// ---- GlobalTextList.TcGTLO
TEXTLIST GlobalTextList
  90 = '\nTwinSAFE'
  12 = '  %s'
  13 = ' %s'
  153 = ' CH1 Test Pulses Active'
  152 = ' CH1 Test Pulses Not Active'
  154 = ' CH2 Test Pulses Active'
  155 = ' CH2 Test Pulses Not Active'
  157 = ' CH3 Test Pulses Active'
  156 = ' CH3 Test Pulses Not Active'
  221 = ' CH32 Test Pulses Not Active'
  159 = ' CH4 Test Pulses Active'
  158 = ' CH4 Test Pulses Not Active'
  222 = ' CH43 Test Pulses Active'
  223 = ' CH5 Test Pulses Active'
  224 = ' CH5 Test Pulses Not Active'
  225 = ' CH6 Test Pulses Active'
  226 = ' CH6 Test Pulses Not Active'
  227 = ' CH7 Test Pulses Active'
  228 = ' CH7 Test Pulses Not Active'
  229 = ' CH8 Test Pulses Active'
  230 = ' CH8 Test Pulses Not Active'
  283 = ' Connections: %s'
  376 = ' CX HW Date: %s'
  374 = ' CX HW Serial#: %s'
  375 = ' CX HW Sn: %s'
  377 = ' CX HW Vers: %s'
  379 = ' CX Image Level: %s'
  378 = ' CX Image Vers: %s'
  373 = ' CX Serial#: %s'
  372 = ' CX: %s'
  286 = ' Groups: %s'
  150 = ' Logic CH1 and CH2: %s'
  151 = ' Logic CH3 and CH4: %s'
  231 = ' Logic CH5 and CH6: %s'
  232 = ' Logic CH7 and CH8: %s'
  143 = ' Mode: %s'
  380 = ' OS Vers: %s'
  371 = ' OS: %s'
  287 = ' Safety FBs: %s'
  43 = '%0.3f'
  363 = '%0i'
  364 = '%0s'
  486 = '%2.1f'
  487 = '%2.1f Hrs'
  362 = '%n'
  365 = '%N'
  11 = '%s'
  509 = '%s v'
  510 = '%sV'
  539 = '(3.300 v Nominal'
  109 = '(3.300 v Nominal)'
  295 = '(5.000 v Nominal)'
  599 = '(ISO 8601) YYYY-MM-DDThh:mm:ss.sTZD'
  101 = '-- External Supply or cross-circuit --\nTHESE ERRORS ARE ONLY ACTIVE IF\nCurrent Measurement is FALSE'
  102 = '-- External Supply or cross-circuit --\nTHESE ERRORS ARE ONLY VALID IF\nCurrent Measurement ACTIVE is FALSE'
  103 = '-- Open Load, I<20mA, I>500mA --\nTHESE ERRORS ARE ONLY VALID IF\nCurrent Measurement ACTIVE is TRUE'
  503 = '. %s'
  35 = '00%s'
  15 = '1'
  16 = '2'
  190 = '2-CHs Eval Error'
  210 = '2CH\nSync\nVel'
  208 = '2CH\nSync Vel'
  209 = '2CH\nSync Vel &\n2CH Encoder'
  203 = '2CH Eval\nError'
  207 = '2CH Sync Vel'
  49 = '2Channel Eval Error'
  17 = '3'
  18 = '4'
  241 = '5'
  443 = '5s'
  242 = '6'
  243 = '7'
  244 = '8'
  161 = '<17.5v'
  165 = '>30.5v'
  160 = '>30v'
  162 = '>320v'
  163 = '>32v'
  508 = 'Actual'
  496 = 'Actual: %s'
  335 = 'AdditionalLink'
  399 = 'ADS Monitor'
  428 = 'ADS Port: %s'
  28 = 'AND#1'
  26 = 'AND#1 Status'
  30 = 'AND#2'
  406 = 'Applic Name: %s'
  297 = 'AX5000 Drive Safety Option: %s'
  343 = 'AX5206'
  316 = 'AX5206 State: %s'
  296 = 'AX5805'
  269 = 'AX5805 Error'
  270 = 'AX5805 OK'
  294 = 'AX5805 Sn: 00%s'
  317 = 'AX5805 State: %s'
  437 = 'AX5808'
  367 = 'Beckhoff Computer and PLC INFO'
  298 = 'Beckhoff EtherCAT Diagnostics 1'
  319 = 'Beckhoff EtherCAT Diagnostics 2'
  442 = 'Beckhoff EtherCAT Diagostics 1'
  449 = 'Beckhoff EtherCAT Diagostics 2'
  502 = 'BIOS: %s'
  490 = 'Boot Count: %s'
  411 = 'Boot Data Loaded'
  408 = 'Boot Data Loaded: %s'
  326 = 'BootStrap'
  176 = 'C\nH\n \n1'
  180 = 'C\nH\n \n2'
  398 = 'Capturing Data'
  94 = 'CH 1'
  137 = 'Ch 1'
  95 = 'CH 2'
  138 = 'Ch 2'
  96 = 'CH 3'
  139 = 'Ch 3'
  97 = 'CH 4'
  140 = 'Ch 4'
  186 = 'Ch 5'
  187 = 'Ch 6'
  188 = 'Ch 7'
  189 = 'Ch 8'
  47 = 'CH1'
  545 = 'Ch1'
  145 = 'CH1 Test Pulses Active'
  144 = 'CH1 Test Pulses Not Active'
  177 = 'CH2'
  546 = 'Ch2'
  146 = 'CH2 Test Pulses Active'
  147 = 'CH2 Test Pulses Not Active'
  178 = 'CH3'
  547 = 'Ch3'
  549 = 'CH3 Test Pulses Active'
  550 = 'CH3 Test Pulses Not Active'
  179 = 'CH4'
  548 = 'Ch4'
  551 = 'CH4 Test Pulses Active'
  552 = 'CH4 Test Pulses Not Active'
  350 = 'Clear\nCRC Errors'
  368 = 'Clear\nFrames Data'
  351 = 'Clear\nLost Frames'
  352 = 'Clear\nTx/Rx Errors'
  347 = 'Clear CRC Errors'
  348 = 'Clear Lost Frames'
  349 = 'Clear Tx/Rx Errors'
  24 = 'COM'
  5 = 'COM Error'
  463 = 'Computer Hardware Specifics'
  465 = 'Computer Software Specifics'
  387 = "Computer's AMSNetID: %s"
  462 = "Computer's AMSNetIDl: %s"
  386 = "Computer'sAMSNetID: %s"
  369 = 'Computer/Controller Specifics'
  21 = 'Connection 1  (EL1904)'
  435 = 'Connection 1 (EL1904)'
  19 = 'Connection 1 State (EL1904)'
  23 = 'Connection 2  (EL2904)'
  436 = 'Connection 2 (EL2904)'
  292 = 'Connections: %s'
  517 = 'CPU Info'
  122 = 'Current Measurement'
  133 = 'Current Measurement Active'
  134 = 'Current Measurement Not Active'
  126 = 'Current Measurement ON'
  500 = 'Currently: %s'
  482 = 'CX Boot Count: %s'
  459 = 'CX HW Date: %s'
  457 = 'CX HW Sn: %s'
  458 = 'CX HW Vers: %s'
  460 = 'CX Image Level: %s'
  388 = 'CX Image Vers: %s'
  483 = 'CX Oper Time - Days: %s'
  484 = 'CX Oper Time - Hrs: %s'
  485 = 'CX Oper Time: %s Days'
  471 = 'CX Prod Date: %D'
  474 = 'CX Prod Date: %M'
  475 = 'CX Prod Date: %m%d%y'
  473 = 'CX Prod Date: %Mdy'
  476 = 'CX Prod Date: %MM-DD-YYYY'
  470 = 'CX Prod Date: %s'
  472 = 'CX Prod Date: %s Mdy'
  478 = 'CX Prod Date: %t[MM DD YYYY]'
  477 = 'CX Prod Date: %t[MM-DD-YYYY]'
  480 = 'CX Prod Date: %t[MM.dd.YYYY]'
  481 = 'CX Prod Date: %t[MM.dd.yyyy]'
  479 = 'CX Prod Date: %t[MM]-%t[dd]-%t[YYYY]'
  468 = 'CX SN: %s'
  469 = 'CX Type: %s'
  389 = 'CX: %s'
  427 = 'Cycle Count: %s'
  424 = 'Cycle Exceeded'
  426 = 'Cycle Exceeded Flag'
  597 = 'Date/Time Presentation: %s'
  534 = 'Default Gateway: %s'
  181 = 'dfgh'
  529 = 'DHCP Flag'
  22 = 'Diagnostic: %s'
  107 = 'DIP SW: %s'
  106 = 'DIP Switch'
  39 = 'DIP Switch Setting'
  248 = 'E-Stop\nComplete'
  33 = 'EDM'
  441 = 'EDM\nFB Error'
  251 = 'EDM FB\nError'
  342 = 'EK1110'
  315 = 'EK1110 State: %s'
  560 = 'EK1122'
  558 = 'EK1122 State: %s'
  340 = 'EL1004'
  310 = 'EL1004 State: %s'
  451 = 'EL1008'
  445 = 'EL1008 State: %s'
  93 = 'EL1904'
  38 = 'EL1904 DIP Switch Setting'
  264 = 'EL1904 Error'
  8 = 'EL1904 Inputs'
  265 = 'EL1904 OK'
  10 = 'EL1904 puts'
  37 = 'EL1904 Serial Number'
  136 = 'EL1904 Sn: 00%s'
  311 = 'EL1904 State: %s'
  341 = 'EL2004'
  312 = 'EL2004 State: %s'
  444 = 'EL2004 State: 5s'
  452 = 'EL2008'
  446 = 'EL2008 State: %s'
  542 = 'EL2901'
  92 = 'EL2904'
  267 = 'EL2904 Error'
  433 = 'EL2904 Inputs'
  268 = 'EL2904 OK'
  9 = 'EL2904 Outputs'
  70 = 'EL2904 Serial Number'
  108 = 'EL2904 Sn: 00%s'
  313 = 'EL2904 State: %s'
  453 = 'EL3002'
  447 = 'EL3002 State: %s'
  559 = 'EL4032'
  556 = 'EL4032 State: %s'
  454 = 'EL4034'
  448 = 'EL4034 State: %s'
  259 = 'EL6900'
  261 = 'EL6900 Error'
  260 = 'EL6900 OK'
  293 = 'EL6900 Sn: 00%s'
  309 = 'EL6900 State: %s'
  282 = 'EL6930'
  262 = 'EL6930 Error'
  263 = 'EL6930 OK'
  182 = 'EL6930 Sn: 00%s'
  314 = 'EL6930 State: %s'
  455 = 'EL7201 #1'
  456 = 'EL7201 #2'
  557 = 'EL7201 State: %s'
  185 = 'EP1908'
  271 = 'EP1908 Error'
  266 = 'EP1908 OK'
  184 = 'EP1908 Sn: 00%s'
  318 = 'EP1908 State: %s'
  247 = 'Error'
  124 = 'Error Ack Active'
  135 = 'Error Ack Not Active'
  71 = 'Error At The Output'
  72 = 'Error At The Output\nExternal Supply or Cross-Circuit'
  169 = 'Error Clear'
  206 = 'Error In Oper Mode'
  29 = 'EStop'
  430 = 'EStop\nComplete'
  438 = 'EStop\nFB'
  439 = 'EStop\nFB Error'
  250 = 'EStop FB\nError'
  0 = 'EStop Reset'
  344 = 'EtherCAT'
  359 = 'EtherCAT\nDiag1'
  360 = 'EtherCAT\nDiag2'
  345 = 'EtherCAT\nDiagnostic 1'
  346 = 'EtherCAT\nDiagnostic 2'
  299 = 'EtherCAT Master Status and Statistics'
  308 = 'EtherCAT Slaves and Working Counter Status'
  358 = 'EtherCAT Working Counter and Slaves Status'
  100 = 'External Supply or cross-circuit\nTHESE ERRORS ARE ONLY ACTIVE IF\nCurrent Measurement is FALSE'
  99 = 'External Supply or cross-circuit\nTHESE ERRORS ARE ONLY ACTIVE IF '
  415 = 'FALSE'
  25 = 'FB'
  6 = 'FB Error'
  543 = 'Features'
  119 = 'Features:'
  423 = 'First Scan'
  425 = 'First Scan Flag'
  586 = 'For CE Only !'
  585 = 'For CE Only !           !'
  584 = 'For CE Only!'
  355 = 'Frames/Sec: %4.0f'
  304 = 'Frames/Sec: %4.1f'
  353 = 'Frames/Sec: %4f'
  205 = 'Frequency\n> 500Hz'
  518 = 'Frequency: %2.3f'
  523 = 'Frequency: %2.3f GHz'
  291 = 'FW: %s'
  67 = 'Go To'
  69 = 'Go To\nEL1904\nDiagnostics'
  68 = 'Go To\nTwinSAFE\nScreen'
  284 = 'Groups: %s'
  75 = 'HI'
  499 = 'Highest: %s'
  289 = 'HW:'
  290 = 'HW: %s'
  511 = 'In Deg C'
  325 = 'Init'
  331 = 'InitCmdError'
  330 = 'InvVPRS'
  532 = 'IP Address: %s'
  410 = 'Keep Outputs ON BP: %s'
  417 = 'Keep Outputs ON Bypass'
  370 = 'Label'
  422 = 'Last Exec Time (100ns incr): %s'
  516 = 'Last Exec Time (in microsec): %5.1f'
  514 = 'Last Exec Time (in microsec): %5.2f'
  515 = 'Last Exec Time (in microsec): %5.3f'
  513 = 'Last Exec Time (in microsec): %s'
  334 = 'LinkMissing'
  332 = 'LinkNotPresent'
  450 = 'Link_w/o_Com'
  333 = 'Link_w/o_Comm'
  76 = 'LO'
  148 = 'Logic CH1 and CH2: %s'
  149 = 'Logic CH3 and CH4: %s'
  34 = 'Logic Terminal Serial Number'
  305 = 'Lost Frames: %i'
  307 = 'Lost Queued Frames: %i'
  498 = 'Lowest: %s'
  531 = 'MAC Address: %s'
  567 = 'Mainboard'
  571 = 'Mainboard and CPU'
  570 = 'Mainboard Info'
  573 = 'Mainboard, CPU, Memory'
  300 = 'Master: %s'
  277 = 'Max Supply Voltage to MC1 Exceeded'
  278 = 'Max Supply Voltage to MC2 Exceeded'
  541 = 'Maximum Supply Voltage to MC1 Exceeded'
  274 = 'Maximum Temperature Exceeded'
  497 = 'Maximum: %s'
  62 = 'MC Temperatures'
  57 = 'MC Temperatures (in Deg C)'
  112 = 'MC Voltages'
  66 = 'MC Voltages (3.300 v Nominal)'
  54 = 'MC Voltages (3.300v Nominal)'
  540 = 'MC1 Actual Temperature: %0.3f v'
  401 = 'MC1 Actual Temperature: %s C'
  104 = 'MC1 Actual Temperature: %s °C'
  110 = 'MC1 Actual Voltage: %0.3f v'
  84 = 'Mc1 COLD!'
  554 = 'MC1 COLD!'
  77 = 'Mc1 HOT!'
  553 = 'MC1 HOT!'
  40 = 'MC1 Temperature'
  42 = 'MC1 Voltage (3.300 Nominal)'
  55 = 'MC1: %0.3f'
  64 = 'MC1: %0.3f v'
  63 = 'MC1: %0.3fv'
  58 = 'MC1: %s'
  60 = 'MC1: %s °C'
  403 = 'MC2 Actual Temperature: %s C'
  105 = 'MC2 Actual Temperature: %s °C'
  402 = 'MC2 Actual Temperature: %s �C'
  111 = 'MC2 Actual Voltage: %0.3f v'
  85 = 'Mc2 COLD!'
  82 = 'Mc2 HOT!'
  555 = 'MC2 HOT!'
  41 = 'MC2 Temperature'
  46 = 'MC2 Voltage (3.300 Nominal)'
  44 = 'MC21 Voltage (3.300 Nominal)'
  56 = 'MC2: %0.3f'
  65 = 'MC2: %0.3f v'
  59 = 'MC2: %s'
  61 = 'MC2: %s °C'
  564 = 'MDP - Mainboard'
  562 = 'MDP - NIC'
  575 = 'Memory Allocated: %s'
  576 = 'Memory Available: %s'
  620 = 'Memory Division: %1.3f GByte'
  583 = 'Memory Division: %s'
  574 = 'Memory Info'
  79 = 'Micro1'
  80 = 'Micro2'
  494 = 'Min: %s'
  495 = 'Minimum: %s'
  544 = 'Mode: %s'
  565 = 'Modulaar Device Profile (MDP)'
  566 = 'Modular Device Profile (MDP)'
  569 = 'Modular Device Profile (MDP) - CX BIOS'
  273 = 'Mximum Temperature Exceeded'
  524 = 'Network Specifics'
  568 = 'NIC'
  530 = 'Nic #1'
  588 = 'NIC #1'
  535 = 'Nic #2'
  589 = 'NIC #2'
  572 = 'NIC and Time'
  587 = 'NIC Info'
  591 = 'NIC, Time'
  528 = 'Nic1 Default Gateway: %s'
  526 = 'Nic1 IP Address: %s'
  525 = 'Nic1 MAC Address: %s'
  527 = 'Nic1 Subnet Mask: %s'
  413 = 'No'
  461 = 'No of PLC Tasks: %s'
  404 = 'No. of PLC Tasks: %s'
  507 = 'Nominal'
  506 = 'Nominal Voltages'
  400 = 'Not Capturing Data'
  301 = 'Number of Configured Slaves: %s'
  303 = 'Number of CRC Errors: %s'
  302 = 'Number of Scanned Slaves: %s'
  416 = 'Old Boot Data'
  409 = 'Old Boot Data: %s'
  407 = 'Online Change Count: %s'
  329 = 'OP'
  491 = 'Oper Time: %s Days'
  393 = 'OS Vers: %s'
  390 = 'OS: %s'
  86 = 'Output COLD!'
  98 = 'Output Errors'
  83 = 'Output HOT!'
  81 = 'OutputBoard'
  50 = 'Pair 1'
  199 = 'Pair 1 / 2'
  214 = 'Pair 1 / 2\n<> Freq'
  213 = 'Pair 1 / 2\nBoth Inactive'
  198 = 'Pair 1/2'
  51 = 'Pair 2'
  200 = 'Pair 3 / 4'
  218 = 'Pair 3 / 4\n<> Freq'
  215 = 'Pair 3 / 4\nBoth Inactive'
  201 = 'Pair 5 / 6'
  219 = 'Pair 5 / 6\n<> Freq'
  216 = 'Pair 5 / 6\nBoth Inactive'
  202 = 'Pair 7 / 8'
  220 = 'Pair 7 / 8\n<> Freq'
  217 = 'Pair 7 / 8\nBoth Inactive'
  191 = 'Pair CH1/CH2'
  192 = 'Pair CH3/CH4'
  193 = 'Pair CH5/CH6'
  194 = 'Pair CH7/CH8'
  405 = 'PLC Proj Name: %s'
  419 = 'PLC Task Name: %s'
  418 = 'PLC Task Specifics'
  336 = 'Port A'
  321 = 'Port A CRC: %s'
  337 = 'Port B'
  322 = 'Port B CRC: %s'
  338 = 'Port C'
  323 = 'Port C CRC: %s'
  339 = 'Port D'
  324 = 'Port D CRC: %s'
  113 = 'Power Rail Voltage Error'
  118 = 'Power Rail Voltage Errors'
  164 = 'Power Rail Voltage Is Above 28.8 v'
  167 = 'Power Rail Voltage Is Above 30.8 v'
  168 = 'Power Rail Voltage Is Below 17.4 v'
  166 = 'Power Rail Voltage Is Below 20.4 v'
  116 = 'Power Rail Voltage Went Above 28.4 v'
  117 = 'Power Rail Voltage Went Above 28.8 v'
  170 = 'Power Rail Voltage Went Above 30.8 v'
  171 = 'Power Rail Voltage Went Below 17.4 v'
  114 = 'Power Rail Voltage Went Below 20.4 v'
  327 = 'PreOP'
  489 = 'Prod Date: %s'
  611 = 'Program Memory Allocated: %1.3f'
  614 = 'Program Memory Allocated: %1.3f GByte'
  608 = 'Program Memory Allocated: %i'
  579 = 'Program Memory Allocated: %s'
  612 = 'Program Memory Available: %1.3f'
  615 = 'Program Memory Available: %1.3f GByte'
  609 = 'Program Memory Available: %i'
  580 = 'Program Memory Available: %s'
  613 = 'Program Memory Used: %1.3f'
  616 = 'Program Memory Used: %1.3f GByte'
  610 = 'Program Memory Used: %i'
  129 = 'Project CRC: %s'
  392 = 'Project Specifics'
  356 = 'Queued Frames/Sec: %4.0f'
  306 = 'Queued Frames/Sec: %4.1f'
  354 = 'Queued Frames/Sec: %4f'
  501 = 'Rev: %s'
  394 = 'Router MAX Memory: %s'
  395 = 'Router Memory Avail: %s'
  396 = 'Router Registered Drivers: %s'
  397 = 'Router Registered Ports: %s'
  391 = 'Router Specifics'
  328 = 'SafeOP'
  255 = 'Safety Connection INFO'
  253 = 'Safety Connections INFO'
  1 = 'Safety Err Ack'
  285 = 'Safety FBs: %s'
  256 = 'Safety Function Block INFO'
  252 = 'Safety Function Blocks INFO'
  173 = 'Safety Group\nErr Ack'
  3 = 'Safety Group \nCOM Error'
  4 = 'Safety Group \nFB Error'
  2 = 'Safety Group COM Error'
  172 = 'Safety Group Err Ack'
  254 = 'Safety Group INFO'
  14 = 'Safety Group Status'
  7 = 'Safety Group1'
   = ''
  434 = 'Safety Group1 Com Err'
  245 = 'Safety Group1 Com Error'
  174 = 'Safety Group1 Communication Error'
  246 = 'Safety Group1 FB Error'
  175 = 'Safety Group1 Function Block Error'
  366 = 'Safety I/O Errors'
  258 = 'Safety I/O INFO'
  212 = 'Safety Mat\nInput Pair\nDisagrees'
  195 = 'Safety Mat\nInput Pair Disagree'
  211 = 'Safety Mat\nTest Pulse\nError'
  196 = 'Safety Mat\nTest Pulse Error'
  204 = 'Safety Mat Input\nPair Disagrees'
  52 = 'Safety Mat Input Pair Disagree'
  141 = 'Safety Mat Test Error'
  142 = 'Safety Mat Test Pulse Error'
  53 = 'Safety Mat Test Pulses Error'
  432 = 'Safety Proj CRC: %0x'
  183 = 'Safety Proj CRC: %s'
  36 = 'Safety Project CRC'
  288 = 'Safety Project INFO:'
  257 = 'Safety Terminal INFO'
  601 = 'Seconds Since 1/1/70: %00.00000000f'
  596 = 'Seconds Since 1/1/70: %s'
  595 = 'Seconds Sinse 1/1/70: %s'
  45 = 'Sensor Test'
  197 = 'Sensor Test\nError'
  48 = 'Sensor Test Error'
  320 = 'Sftw Rev: %s'
  592 = 'SMTP Server: %s'
  488 = 'SN: %s'
  607 = 'SNTP Refresh in Minutes: %0.2f'
  600 = 'SNTP Refresh: %0.00f'
  604 = 'SNTP Refresh: %0.2f'
  594 = 'SNTP Refresh: %s'
  593 = 'SNTP Server: %s'
  120 = 'Standard Outputs'
  131 = 'Standard Outputs Active'
  127 = 'Standard Outputs Enabled'
  130 = 'Standard Outputs Not Active'
  121 = 'Standard Outputs:'
  20 = 'State: %s'
  27 = 'Status: %s'
  577 = 'Storage Allocated: %s'
  578 = 'Storage Available: %s'
  617 = 'Storage Memory Allocated: %1.3f GByte'
  581 = 'Storage Memory Allocated: %s'
  618 = 'Storage Memory Available: %1.3f GByte'
  582 = 'Storage Memory Available: %s'
  619 = 'Storage Memory Used: %1.3f GByte'
  128 = 'Store Code: %s'
  533 = 'Subnet Mask: %s'
  74 = 'Supply Voltage Error'
  73 = 'Supply Voltage Error\nVoltage Hi     Voltage Lo'
  538 = 'SW: %s'
  89 = 'T-Diff Between MCs Too Large!'
  561 = 'T-Diff between MCs Too Large!'
  88 = 'T-Diff on MC Too Large!'
  421 = 'Task Cycle Time (100ns incr): %s'
  537 = 'Task Cycle Time (in microsec): %5.0f'
  536 = 'Task Cycle Time (in microsec): %5.1f'
  512 = 'Task Cycle Time (in microsec): %s'
  420 = 'Task Cycle Time: %s'
  429 = 'Task Priority: %s'
  384 = 'Tc Build: %s'
  385 = 'Tc Level: %s'
  382 = 'Tc Maj Vers: %s'
  383 = 'Tc Min Vers: %s'
  381 = 'Tc Vers: %s'
  87 = 'Temp Diff on MC Too Large!'
  272 = 'Temperature\nErrors'
  276 = 'Temperature Difference Between\nMeasuring Points Exceeded'
  78 = 'Temperature Errors'
  275 = 'Temperature Fell Below Minimum'
  520 = 'Temperature: %s'
  521 = 'Temperature: %s DegC'
  492 = 'Temperatures'
  493 = 'Temperatures in DegC'
  504 = 'Temps in DegC'
  123 = 'Test Pulses'
  125 = 'Test Pulses Active'
  132 = 'Test Pulses Not Active'
  590 = 'Time Info'
  249 = 'Timer\nComplete'
  598 = 'Timezone: %s'
  32 = 'TOF'
  440 = 'TOF\nComplete'
  31 = 'TON'
  431 = 'TON\nComplete'
  414 = 'TRUE'
  361 = 'TwinCAT\nINFO'
  563 = 'TwinCAT INFO'
  464 = 'TwinCAT Project Specifics'
  466 = 'TwinCAT Router Specifics'
  91 = 'TwinSAFE'
  467 = 'Type: %s'
  519 = 'Usage: %s'
  522 = 'Usage: %s %'
  233 = 'VelLIM1: %s'
  234 = 'VelLIM2: %s'
  235 = 'VelLIM3: %s'
  236 = 'VelLIM4: %s'
  237 = 'VelLIM5: %s'
  238 = 'VelLIM6: %s'
  239 = 'VelLIM7: %s'
  240 = 'VelLIM8: %s'
  115 = 'Voltage Errors'
  280 = 'Voltage Fell Below\nMin Supply Voltage to MC1'
  281 = 'Voltage Fell Below\nMin Supply Voltage to MC2'
  279 = 'Voltage Fell Below Min Supply Voltage to MC1'
  505 = 'Voltages'
  357 = 'W/C'
  603 = 'Years Since 1/1/70: %0.00000000f'
  605 = 'Years Since 1/1/70: %0.10f'
  606 = 'Years Since 1/1/70: %0.8f'
  602 = 'Years Since 1/1/70: %00.00000000f'
  412 = 'Yes'
END_TEXTLIST

// ---- VISUs/AX5805_Specific_Diagnostics.TcVIS
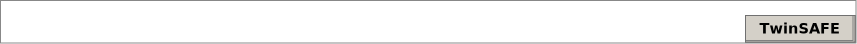
VISUALIZATION AX5805_Specific_Diagnostics  // 857x44
    Button (745,15 110x27), "TwinSAFE"
        OnMouseClick: change screen: TwinSAFE
        OnMouseUp: execute { g_xHMI_ErrAckPB := FALSE ; }
END_VISUALIZATION

// ---- VISUs/AX5805_Specific_Diagnostics.TcVIS
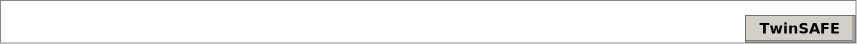
VISUALIZATION AX5805_Specific_Diagnostics  // 857x44
    Button (745,15 110x27), "TwinSAFE"
        OnMouseClick: change screen: TwinSAFE
        OnMouseUp: execute { g_xHMI_ErrAckPB := FALSE ; }
END_VISUALIZATION

// ---- VISUs/AX5805_Specific_Diagnostics.TcVIS
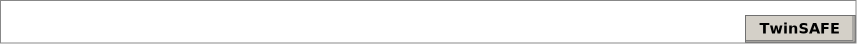
VISUALIZATION AX5805_Specific_Diagnostics  // 857x44
    Button (745,15 110x27), "TwinSAFE"
        OnMouseClick: change screen: TwinSAFE
        OnMouseUp: execute { g_xHMI_ErrAckPB := FALSE ; }
END_VISUALIZATION

// ---- VISUs/EL2904_Specific_Diagnostics.TcVIS
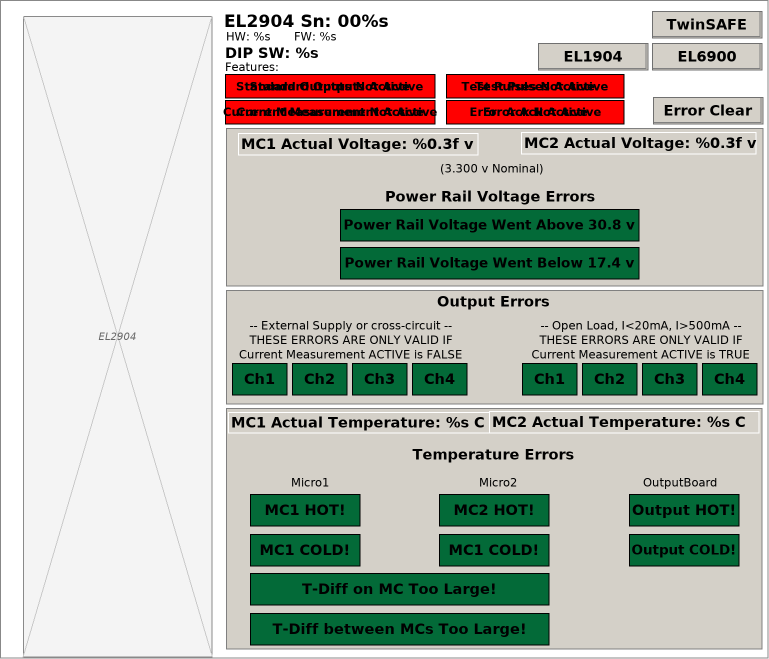
VISUALIZATION EL2904_Specific_Diagnostics  // 769x659
    Button (652,11 110x27), "TwinSAFE"
        OnMouseClick: change screen: TwinSAFE
    Button (652,43 110x27), "EL6900"
        OnMouseClick: change screen: EL6900_Specific_Diagnostics
    Button (538,43 110x27), "EL1904"
        OnMouseClick: change screen: EL1904_Specific_Diagnostics
    Image (23,16 189x641), image: EL2904
    Rectangle (221,10 275x22), "EL2904 Sn: 00%s", text variable: g_dwHMI_EL2904Sn
    Rectangle (223,28 65x17), "HW: %s", text variable: g_sHMI_EL2904_HWvers
    Rectangle (291,28 65x17), "FW: %s", text variable: g_sHMI_EL2904_FWvers
    Rectangle (222,45 164x16), "DIP SW: %s", text variable: g_wHMI_EL2904DSw
    Label (222,59 88x16), "Features:"
    Button (653,97 110x27), "Error Clear"
        OnMouseUp: execute { g_xHMI_EL2904_ErrClearPB := FALSE ; }
        OnMouseDown: execute { g_xHMI_EL2904_ErrClearPB := TRUE ; }
    Rectangle (226,128 537x158)
    Label (433,161 118x15), "(3.300 v Nominal)"
    Rectangle (238,133 240x22), "MC1 Actual Voltage: %0.3f v", text variable: g_wHMI_EL2904PriMC_Volts
    Rectangle (521,132 235x22), "MC2 Actual Voltage: %0.3f v", text variable: g_wHMI_EL2904SecMC_Volts
    Rectangle (226,290 537x114)
    Rectangle (226,408 536x241)
    Rectangle (228,412 264x21), "MC1 Actual Temperature: %s C", text variable: g_wHMI_EL2904PriMCTemp
    Rectangle (489,411 270x22), "MC2 Actual Temperature: %s C", text variable: g_wHMI_EL2904SecMCTemp
    Label (280,474 61x17), "Micro1"
    Label (402,440 183x29), "Temperature Errors"
    Label (225,311 252x58), "-- External Supply or cross-circuit -- THESE ERRORS ARE ONLY VALID IF Current Measurement ACTIVE is FALSE"
    Label (376,185 228x23), "Power Rail Voltage Errors"
    Label (429,287 129x29), "Output Errors"
    Rectangle (340,209 299x32), "Power Rail Voltage Went Above 30.8 v", colour toggle: g_xHMI_EL2904_PwrRailVoltageHi
    Rectangle (340,247 299x32), "Power Rail Voltage Went Below 17.4 v", colour toggle: g_xHMI_EL2904_PwrRailVoltageLo
    Label (515,311 252x58), "-- Open Load, I<20mA, I>500mA -- THESE ERRORS ARE ONLY VALID IF Current Measurement ACTIVE is TRUE"
    Rectangle (232,363 55x32), "Ch1", colour toggle: g_xHMI_EL2904_ExtSup_CrossCirErr_Out1
    Rectangle (292,363 55x32), "Ch2", colour toggle: g_xHMI_EL2904_ExtSup_CrossCirErr_Out2
    Rectangle (352,363 55x32), "Ch3", colour toggle: g_xHMI_EL2904_ExtSup_CrossCirErr_Out3
    Rectangle (412,363 55x32), "Ch4", colour toggle: g_xHMI_EL2904_ExtSup_CrossCirErr_Out4
    Rectangle (522,363 55x32), "Ch1", colour toggle: g_xHMI_EL2904_OutLoadErr_Out1
    Rectangle (582,363 55x32), "Ch2", colour toggle: g_xHMI_EL2904_OutLoadErr_Out2
    Rectangle (642,363 55x32), "Ch3", colour toggle: g_xHMI_EL2904_OutLoadErr_Out3
    Rectangle (702,363 55x32), "Ch4", colour toggle: g_xHMI_EL2904_OutLoadErr_Out4
    Label (468,474 61x17), "Micro2"
    Label (633,474 95x17), "OutputBoard"
    Rectangle (250,494 110x32), "MC1 HOT!", colour toggle: g_xHMI_EL2904_TempErr_OTMc1
    Rectangle (250,534 110x32), "MC1 COLD!", colour toggle: g_xHMI_EL2904_TempErr_UTMc1
    Rectangle (439,494 110x32), "MC2 HOT!", colour toggle: g_xHMI_EL2904_TempErr_OTMc2
    Rectangle (439,534 110x32), "MC1 COLD!", colour toggle: g_xHMI_EL2904_TempErr_UTMc2
    Rectangle (629,494 110x32), "Output HOT!", colour toggle: g_xHMI_EL2904_TempErr_OTOutBoard
    Rectangle (629,534 110x32), "Output COLD!", colour toggle: g_xHMI_EL2904_TempErr_UTOutBoard
    Rectangle (250,573 299x32), "T-Diff on MC Too Large!", colour toggle: g_xHMI_EL2904_TempErr_DiffOnBoard
    Rectangle (250,613 299x32), "T-Diff between MCs Too Large!", colour toggle: g_xHMI_EL2904_TempErr_DiffBetweenMc1Mc2
    Rectangle (225,74 210x24), colour toggle: g_xHMI_EL2904_StandardOuts
    Rectangle (446,74 178x24), colour toggle: g_xHMI_EL2904_TestPulses
    Rectangle (225,100 210x24), colour toggle: g_xHMI_EL2904_CurrentMeas
    Rectangle (446,100 178x24), colour toggle: g_xHMI_EL2904_ErrAck
    Group (241,75 178x23)
        Label (0,0 178x23), "Standard Outputs Not Active", invisible if: g_xHMI_EL2904_StandardOuts
        Label (0,0 178x23), "Standard Outputs Active", invisible if: not g_xHMI_EL2904_StandardOuts
    Group (446,75 178x23)
        Label (0,0 178x23), "Test Pulses Not Active", invisible if: g_xHMI_EL2904_TestPulses
        Label (0,0 178x23), "Test Pulses Active", invisible if: not g_xHMI_EL2904_TestPulses
    Group (226,97 209x30)
        Label (0,0 209x30), "Current Measurement Not Active", invisible if: g_xHMI_EL2904_CurrentMeas
        Label (6,0 197x30), "Current Measurement Active", invisible if: not g_xHMI_EL2904_CurrentMeas
    Group (462,97 147x30)
        Label (0,0 147x30), "Error Ack Not Active", invisible if: g_xHMI_EL2904_ErrAck
        Label (0,0 147x30), "Error Ack Active", invisible if: not g_xHMI_EL2904_ErrAck
END_VISUALIZATION

// ---- VISUs/EL2904_Specific_Diagnostics.TcVIS
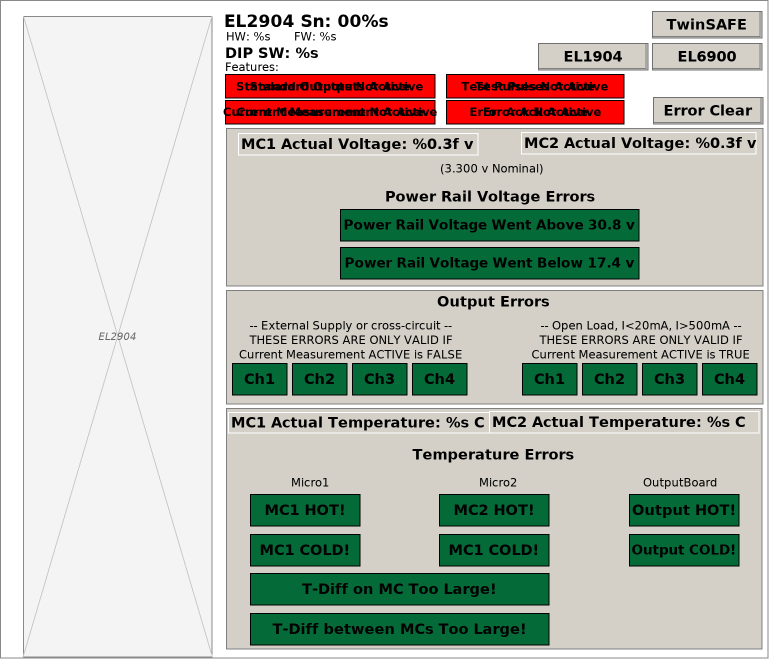
VISUALIZATION EL2904_Specific_Diagnostics  // 769x659
    Button (652,11 110x27), "TwinSAFE"
        OnMouseClick: change screen: TwinSAFE
    Button (652,43 110x27), "EL6900"
        OnMouseClick: change screen: EL6900_Specific_Diagnostics
    Button (538,43 110x27), "EL1904"
        OnMouseClick: change screen: EL1904_Specific_Diagnostics
    Image (23,16 189x641), image: EL2904
    Rectangle (221,10 275x22), "EL2904 Sn: 00%s", text variable: g_dwHMI_EL2904Sn
    Rectangle (223,28 65x17), "HW: %s", text variable: g_sHMI_EL2904_HWvers
    Rectangle (291,28 65x17), "FW: %s", text variable: g_sHMI_EL2904_FWvers
    Rectangle (222,45 164x16), "DIP SW: %s", text variable: g_wHMI_EL2904DSw
    Label (222,59 88x16), "Features:"
    Button (653,97 110x27), "Error Clear"
        OnMouseUp: execute { g_xHMI_EL2904_ErrClearPB := FALSE ; }
        OnMouseDown: execute { g_xHMI_EL2904_ErrClearPB := TRUE ; }
    Rectangle (226,128 537x158)
    Label (433,161 118x15), "(3.300 v Nominal)"
    Rectangle (238,133 240x22), "MC1 Actual Voltage: %0.3f v", text variable: g_wHMI_EL2904PriMC_Volts
    Rectangle (521,132 235x22), "MC2 Actual Voltage: %0.3f v", text variable: g_wHMI_EL2904SecMC_Volts
    Rectangle (226,290 537x114)
    Rectangle (226,408 536x241)
    Rectangle (228,412 264x21), "MC1 Actual Temperature: %s C", text variable: g_wHMI_EL2904PriMCTemp
    Rectangle (489,411 270x22), "MC2 Actual Temperature: %s C", text variable: g_wHMI_EL2904SecMCTemp
    Label (280,474 61x17), "Micro1"
    Label (402,440 183x29), "Temperature Errors"
    Label (225,311 252x58), "-- External Supply or cross-circuit -- THESE ERRORS ARE ONLY VALID IF Current Measurement ACTIVE is FALSE"
    Label (376,185 228x23), "Power Rail Voltage Errors"
    Label (429,287 129x29), "Output Errors"
    Rectangle (340,209 299x32), "Power Rail Voltage Went Above 30.8 v", colour toggle: g_xHMI_EL2904_PwrRailVoltageHi
    Rectangle (340,247 299x32), "Power Rail Voltage Went Below 17.4 v", colour toggle: g_xHMI_EL2904_PwrRailVoltageLo
    Label (515,311 252x58), "-- Open Load, I<20mA, I>500mA -- THESE ERRORS ARE ONLY VALID IF Current Measurement ACTIVE is TRUE"
    Rectangle (232,363 55x32), "Ch1", colour toggle: g_xHMI_EL2904_ExtSup_CrossCirErr_Out1
    Rectangle (292,363 55x32), "Ch2", colour toggle: g_xHMI_EL2904_ExtSup_CrossCirErr_Out2
    Rectangle (352,363 55x32), "Ch3", colour toggle: g_xHMI_EL2904_ExtSup_CrossCirErr_Out3
    Rectangle (412,363 55x32), "Ch4", colour toggle: g_xHMI_EL2904_ExtSup_CrossCirErr_Out4
    Rectangle (522,363 55x32), "Ch1", colour toggle: g_xHMI_EL2904_OutLoadErr_Out1
    Rectangle (582,363 55x32), "Ch2", colour toggle: g_xHMI_EL2904_OutLoadErr_Out2
    Rectangle (642,363 55x32), "Ch3", colour toggle: g_xHMI_EL2904_OutLoadErr_Out3
    Rectangle (702,363 55x32), "Ch4", colour toggle: g_xHMI_EL2904_OutLoadErr_Out4
    Label (468,474 61x17), "Micro2"
    Label (633,474 95x17), "OutputBoard"
    Rectangle (250,494 110x32), "MC1 HOT!", colour toggle: g_xHMI_EL2904_TempErr_OTMc1
    Rectangle (250,534 110x32), "MC1 COLD!", colour toggle: g_xHMI_EL2904_TempErr_UTMc1
    Rectangle (439,494 110x32), "MC2 HOT!", colour toggle: g_xHMI_EL2904_TempErr_OTMc2
    Rectangle (439,534 110x32), "MC1 COLD!", colour toggle: g_xHMI_EL2904_TempErr_UTMc2
    Rectangle (629,494 110x32), "Output HOT!", colour toggle: g_xHMI_EL2904_TempErr_OTOutBoard
    Rectangle (629,534 110x32), "Output COLD!", colour toggle: g_xHMI_EL2904_TempErr_UTOutBoard
    Rectangle (250,573 299x32), "T-Diff on MC Too Large!", colour toggle: g_xHMI_EL2904_TempErr_DiffOnBoard
    Rectangle (250,613 299x32), "T-Diff between MCs Too Large!", colour toggle: g_xHMI_EL2904_TempErr_DiffBetweenMc1Mc2
    Rectangle (225,74 210x24), colour toggle: g_xHMI_EL2904_StandardOuts
    Rectangle (446,74 178x24), colour toggle: g_xHMI_EL2904_TestPulses
    Rectangle (225,100 210x24), colour toggle: g_xHMI_EL2904_CurrentMeas
    Rectangle (446,100 178x24), colour toggle: g_xHMI_EL2904_ErrAck
    Group (241,75 178x23)
        Label (0,0 178x23), "Standard Outputs Not Active", invisible if: g_xHMI_EL2904_StandardOuts
        Label (0,0 178x23), "Standard Outputs Active", invisible if: not g_xHMI_EL2904_StandardOuts
    Group (446,75 178x23)
        Label (0,0 178x23), "Test Pulses Not Active", invisible if: g_xHMI_EL2904_TestPulses
        Label (0,0 178x23), "Test Pulses Active", invisible if: not g_xHMI_EL2904_TestPulses
    Group (226,97 209x30)
        Label (0,0 209x30), "Current Measurement Not Active", invisible if: g_xHMI_EL2904_CurrentMeas
        Label (6,0 197x30), "Current Measurement Active", invisible if: not g_xHMI_EL2904_CurrentMeas
    Group (462,97 147x30)
        Label (0,0 147x30), "Error Ack Not Active", invisible if: g_xHMI_EL2904_ErrAck
        Label (0,0 147x30), "Error Ack Active", invisible if: not g_xHMI_EL2904_ErrAck
END_VISUALIZATION

// ---- VISUs/EL2904_Specific_Diagnostics.TcVIS
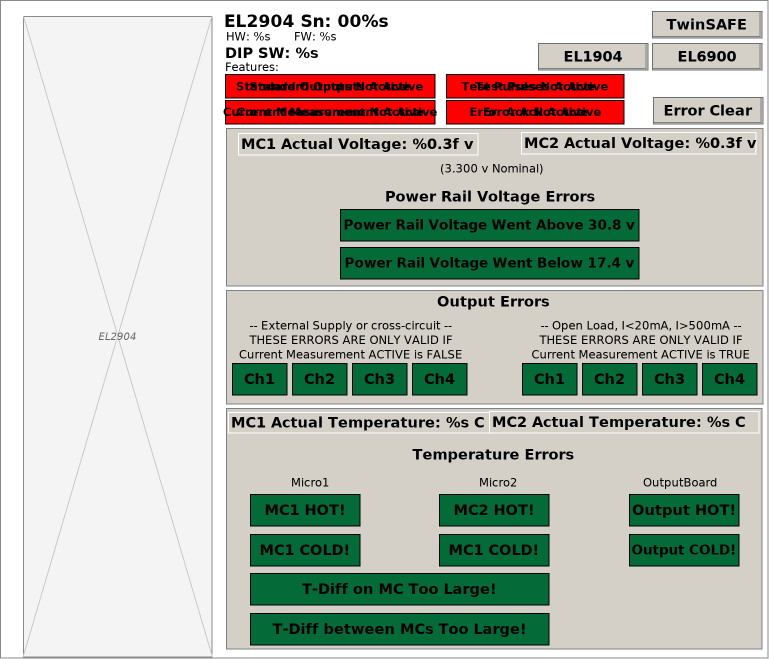
VISUALIZATION EL2904_Specific_Diagnostics  // 769x659
    Button (652,11 110x27), "TwinSAFE"
        OnMouseClick: change screen: TwinSAFE
    Button (652,43 110x27), "EL6900"
        OnMouseClick: change screen: EL6900_Specific_Diagnostics
    Button (538,43 110x27), "EL1904"
        OnMouseClick: change screen: EL1904_Specific_Diagnostics
    Image (23,16 189x641), image: EL2904
    Rectangle (221,10 275x22), "EL2904 Sn: 00%s", text variable: g_dwHMI_EL2904Sn
    Rectangle (223,28 65x17), "HW: %s", text variable: g_sHMI_EL2904_HWvers
    Rectangle (291,28 65x17), "FW: %s", text variable: g_sHMI_EL2904_FWvers
    Rectangle (222,45 164x16), "DIP SW: %s", text variable: g_wHMI_EL2904DSw
    Label (222,59 88x16), "Features:"
    Button (653,97 110x27), "Error Clear"
        OnMouseUp: execute { g_xHMI_EL2904_ErrClearPB := FALSE ; }
        OnMouseDown: execute { g_xHMI_EL2904_ErrClearPB := TRUE ; }
    Rectangle (226,128 537x158)
    Label (433,161 118x15), "(3.300 v Nominal)"
    Rectangle (238,133 240x22), "MC1 Actual Voltage: %0.3f v", text variable: g_wHMI_EL2904PriMC_Volts
    Rectangle (521,132 235x22), "MC2 Actual Voltage: %0.3f v", text variable: g_wHMI_EL2904SecMC_Volts
    Rectangle (226,290 537x114)
    Rectangle (226,408 536x241)
    Rectangle (228,412 264x21), "MC1 Actual Temperature: %s C", text variable: g_wHMI_EL2904PriMCTemp
    Rectangle (489,411 270x22), "MC2 Actual Temperature: %s C", text variable: g_wHMI_EL2904SecMCTemp
    Label (280,474 61x17), "Micro1"
    Label (402,440 183x29), "Temperature Errors"
    Label (225,311 252x58), "-- External Supply or cross-circuit -- THESE ERRORS ARE ONLY VALID IF Current Measurement ACTIVE is FALSE"
    Label (376,185 228x23), "Power Rail Voltage Errors"
    Label (429,287 129x29), "Output Errors"
    Rectangle (340,209 299x32), "Power Rail Voltage Went Above 30.8 v", colour toggle: g_xHMI_EL2904_PwrRailVoltageHi
    Rectangle (340,247 299x32), "Power Rail Voltage Went Below 17.4 v", colour toggle: g_xHMI_EL2904_PwrRailVoltageLo
    Label (515,311 252x58), "-- Open Load, I<20mA, I>500mA -- THESE ERRORS ARE ONLY VALID IF Current Measurement ACTIVE is TRUE"
    Rectangle (232,363 55x32), "Ch1", colour toggle: g_xHMI_EL2904_ExtSup_CrossCirErr_Out1
    Rectangle (292,363 55x32), "Ch2", colour toggle: g_xHMI_EL2904_ExtSup_CrossCirErr_Out2
    Rectangle (352,363 55x32), "Ch3", colour toggle: g_xHMI_EL2904_ExtSup_CrossCirErr_Out3
    Rectangle (412,363 55x32), "Ch4", colour toggle: g_xHMI_EL2904_ExtSup_CrossCirErr_Out4
    Rectangle (522,363 55x32), "Ch1", colour toggle: g_xHMI_EL2904_OutLoadErr_Out1
    Rectangle (582,363 55x32), "Ch2", colour toggle: g_xHMI_EL2904_OutLoadErr_Out2
    Rectangle (642,363 55x32), "Ch3", colour toggle: g_xHMI_EL2904_OutLoadErr_Out3
    Rectangle (702,363 55x32), "Ch4", colour toggle: g_xHMI_EL2904_OutLoadErr_Out4
    Label (468,474 61x17), "Micro2"
    Label (633,474 95x17), "OutputBoard"
    Rectangle (250,494 110x32), "MC1 HOT!", colour toggle: g_xHMI_EL2904_TempErr_OTMc1
    Rectangle (250,534 110x32), "MC1 COLD!", colour toggle: g_xHMI_EL2904_TempErr_UTMc1
    Rectangle (439,494 110x32), "MC2 HOT!", colour toggle: g_xHMI_EL2904_TempErr_OTMc2
    Rectangle (439,534 110x32), "MC1 COLD!", colour toggle: g_xHMI_EL2904_TempErr_UTMc2
    Rectangle (629,494 110x32), "Output HOT!", colour toggle: g_xHMI_EL2904_TempErr_OTOutBoard
    Rectangle (629,534 110x32), "Output COLD!", colour toggle: g_xHMI_EL2904_TempErr_UTOutBoard
    Rectangle (250,573 299x32), "T-Diff on MC Too Large!", colour toggle: g_xHMI_EL2904_TempErr_DiffOnBoard
    Rectangle (250,613 299x32), "T-Diff between MCs Too Large!", colour toggle: g_xHMI_EL2904_TempErr_DiffBetweenMc1Mc2
    Rectangle (225,74 210x24), colour toggle: g_xHMI_EL2904_StandardOuts
    Rectangle (446,74 178x24), colour toggle: g_xHMI_EL2904_TestPulses
    Rectangle (225,100 210x24), colour toggle: g_xHMI_EL2904_CurrentMeas
    Rectangle (446,100 178x24), colour toggle: g_xHMI_EL2904_ErrAck
    Group (241,75 178x23)
        Label (0,0 178x23), "Standard Outputs Not Active", invisible if: g_xHMI_EL2904_StandardOuts
        Label (0,0 178x23), "Standard Outputs Active", invisible if: not g_xHMI_EL2904_StandardOuts
    Group (446,75 178x23)
        Label (0,0 178x23), "Test Pulses Not Active", invisible if: g_xHMI_EL2904_TestPulses
        Label (0,0 178x23), "Test Pulses Active", invisible if: not g_xHMI_EL2904_TestPulses
    Group (226,97 209x30)
        Label (0,0 209x30), "Current Measurement Not Active", invisible if: g_xHMI_EL2904_CurrentMeas
        Label (6,0 197x30), "Current Measurement Active", invisible if: not g_xHMI_EL2904_CurrentMeas
    Group (462,97 147x30)
        Label (0,0 147x30), "Error Ack Not Active", invisible if: g_xHMI_EL2904_ErrAck
        Label (0,0 147x30), "Error Ack Active", invisible if: not g_xHMI_EL2904_ErrAck
END_VISUALIZATION

// ---- VISUs/EL2904_Specific_Diagnostics.TcVIS
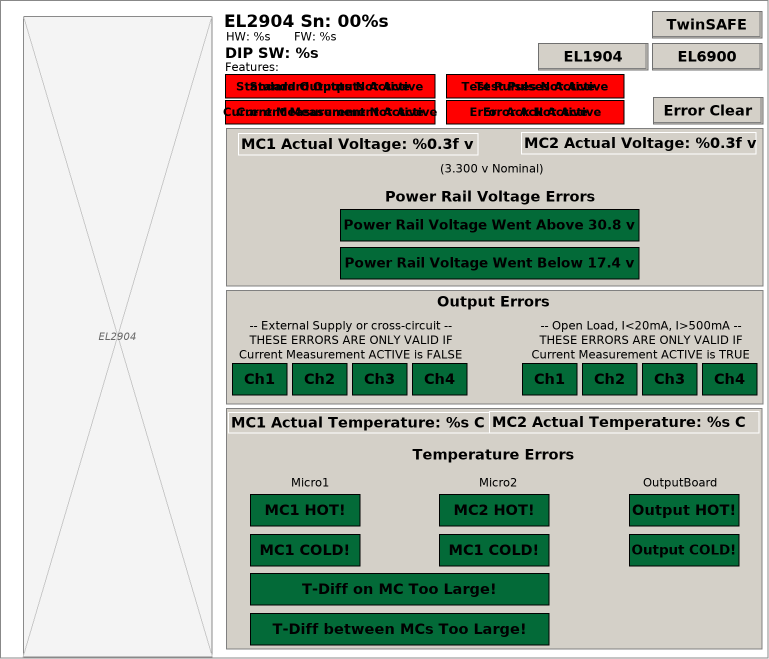
VISUALIZATION EL2904_Specific_Diagnostics  // 769x659
    Button (652,11 110x27), "TwinSAFE"
        OnMouseClick: change screen: TwinSAFE
    Button (652,43 110x27), "EL6900"
        OnMouseClick: change screen: EL6900_Specific_Diagnostics
    Button (538,43 110x27), "EL1904"
        OnMouseClick: change screen: EL1904_Specific_Diagnostics
    Image (23,16 189x641), image: EL2904
    Rectangle (221,10 275x22), "EL2904 Sn: 00%s", text variable: g_dwHMI_EL2904Sn
    Rectangle (223,28 65x17), "HW: %s", text variable: g_sHMI_EL2904_HWvers
    Rectangle (291,28 65x17), "FW: %s", text variable: g_sHMI_EL2904_FWvers
    Rectangle (222,45 164x16), "DIP SW: %s", text variable: g_wHMI_EL2904DSw
    Label (222,59 88x16), "Features:"
    Button (653,97 110x27), "Error Clear"
        OnMouseUp: execute { g_xHMI_EL2904_ErrClearPB := FALSE ; }
        OnMouseDown: execute { g_xHMI_EL2904_ErrClearPB := TRUE ; }
    Rectangle (226,128 537x158)
    Label (433,161 118x15), "(3.300 v Nominal)"
    Rectangle (238,133 240x22), "MC1 Actual Voltage: %0.3f v", text variable: g_wHMI_EL2904PriMC_Volts
    Rectangle (521,132 235x22), "MC2 Actual Voltage: %0.3f v", text variable: g_wHMI_EL2904SecMC_Volts
    Rectangle (226,290 537x114)
    Rectangle (226,408 536x241)
    Rectangle (228,412 264x21), "MC1 Actual Temperature: %s C", text variable: g_wHMI_EL2904PriMCTemp
    Rectangle (489,411 270x22), "MC2 Actual Temperature: %s C", text variable: g_wHMI_EL2904SecMCTemp
    Label (280,474 61x17), "Micro1"
    Label (402,440 183x29), "Temperature Errors"
    Label (225,311 252x58), "-- External Supply or cross-circuit -- THESE ERRORS ARE ONLY VALID IF Current Measurement ACTIVE is FALSE"
    Label (376,185 228x23), "Power Rail Voltage Errors"
    Label (429,287 129x29), "Output Errors"
    Rectangle (340,209 299x32), "Power Rail Voltage Went Above 30.8 v", colour toggle: g_xHMI_EL2904_PwrRailVoltageHi
    Rectangle (340,247 299x32), "Power Rail Voltage Went Below 17.4 v", colour toggle: g_xHMI_EL2904_PwrRailVoltageLo
    Label (515,311 252x58), "-- Open Load, I<20mA, I>500mA -- THESE ERRORS ARE ONLY VALID IF Current Measurement ACTIVE is TRUE"
    Rectangle (232,363 55x32), "Ch1", colour toggle: g_xHMI_EL2904_ExtSup_CrossCirErr_Out1
    Rectangle (292,363 55x32), "Ch2", colour toggle: g_xHMI_EL2904_ExtSup_CrossCirErr_Out2
    Rectangle (352,363 55x32), "Ch3", colour toggle: g_xHMI_EL2904_ExtSup_CrossCirErr_Out3
    Rectangle (412,363 55x32), "Ch4", colour toggle: g_xHMI_EL2904_ExtSup_CrossCirErr_Out4
    Rectangle (522,363 55x32), "Ch1", colour toggle: g_xHMI_EL2904_OutLoadErr_Out1
    Rectangle (582,363 55x32), "Ch2", colour toggle: g_xHMI_EL2904_OutLoadErr_Out2
    Rectangle (642,363 55x32), "Ch3", colour toggle: g_xHMI_EL2904_OutLoadErr_Out3
    Rectangle (702,363 55x32), "Ch4", colour toggle: g_xHMI_EL2904_OutLoadErr_Out4
    Label (468,474 61x17), "Micro2"
    Label (633,474 95x17), "OutputBoard"
    Rectangle (250,494 110x32), "MC1 HOT!", colour toggle: g_xHMI_EL2904_TempErr_OTMc1
    Rectangle (250,534 110x32), "MC1 COLD!", colour toggle: g_xHMI_EL2904_TempErr_UTMc1
    Rectangle (439,494 110x32), "MC2 HOT!", colour toggle: g_xHMI_EL2904_TempErr_OTMc2
    Rectangle (439,534 110x32), "MC1 COLD!", colour toggle: g_xHMI_EL2904_TempErr_UTMc2
    Rectangle (629,494 110x32), "Output HOT!", colour toggle: g_xHMI_EL2904_TempErr_OTOutBoard
    Rectangle (629,534 110x32), "Output COLD!", colour toggle: g_xHMI_EL2904_TempErr_UTOutBoard
    Rectangle (250,573 299x32), "T-Diff on MC Too Large!", colour toggle: g_xHMI_EL2904_TempErr_DiffOnBoard
    Rectangle (250,613 299x32), "T-Diff between MCs Too Large!", colour toggle: g_xHMI_EL2904_TempErr_DiffBetweenMc1Mc2
    Rectangle (225,74 210x24), colour toggle: g_xHMI_EL2904_StandardOuts
    Rectangle (446,74 178x24), colour toggle: g_xHMI_EL2904_TestPulses
    Rectangle (225,100 210x24), colour toggle: g_xHMI_EL2904_CurrentMeas
    Rectangle (446,100 178x24), colour toggle: g_xHMI_EL2904_ErrAck
    Group (241,75 178x23)
        Label (0,0 178x23), "Standard Outputs Not Active", invisible if: g_xHMI_EL2904_StandardOuts
        Label (0,0 178x23), "Standard Outputs Active", invisible if: not g_xHMI_EL2904_StandardOuts
    Group (446,75 178x23)
        Label (0,0 178x23), "Test Pulses Not Active", invisible if: g_xHMI_EL2904_TestPulses
        Label (0,0 178x23), "Test Pulses Active", invisible if: not g_xHMI_EL2904_TestPulses
    Group (226,97 209x30)
        Label (0,0 209x30), "Current Measurement Not Active", invisible if: g_xHMI_EL2904_CurrentMeas
        Label (6,0 197x30), "Current Measurement Active", invisible if: not g_xHMI_EL2904_CurrentMeas
    Group (462,97 147x30)
        Label (0,0 147x30), "Error Ack Not Active", invisible if: g_xHMI_EL2904_ErrAck
        Label (0,0 147x30), "Error Ack Active", invisible if: not g_xHMI_EL2904_ErrAck
END_VISUALIZATION

// ---- VISUs/EL6900_Specific_Diagnostics.TcVIS
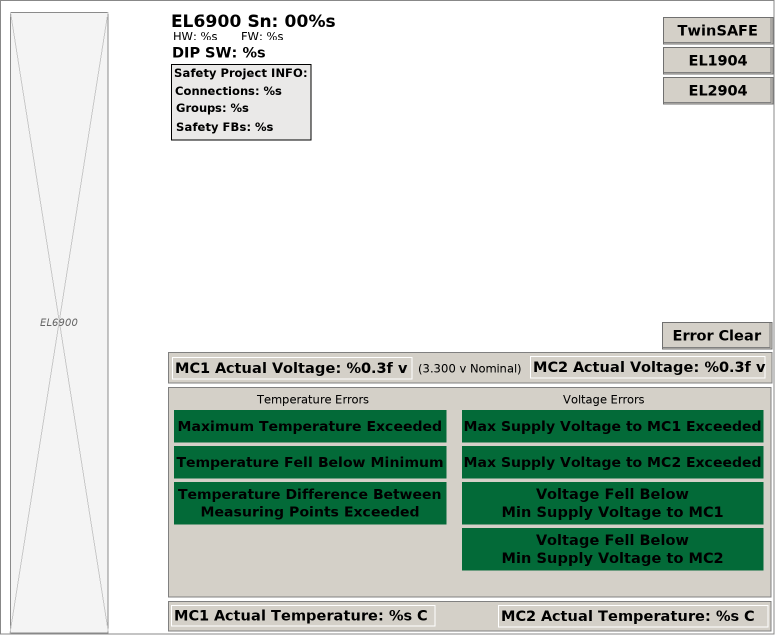
VISUALIZATION EL6900_Specific_Diagnostics  // 775x635
    Button (663,17 110x27), "TwinSAFE"
        OnMouseClick: change screen: TwinSAFE
    Button (663,47 110x27), "EL1904"
        OnMouseClick: change screen: EL1904_Specific_Diagnostics
    Button (663,77 110x27), "EL2904"
        OnMouseClick: change screen: EL2904_Specific_Diagnostics
    Image (10,12 98x621), image: EL6900
    Rectangle (168,10 275x22), "EL6900 Sn: 00%s", text variable: g_dwHMI_EL6900Sn
    Rectangle (170,28 65x17), "HW: %s", text variable: g_sHMI_EL6900_HWvers
    Rectangle (238,28 65x17), "FW: %s", text variable: g_sHMI_EL6900_FWvers
    Rectangle (169,40 136x25), "DIP SW: %s", text variable: g_wHMI_EL6900DSw
    Group (171,62 140x78)
        Rectangle (0,2 140x76)
        Rectangle (1,17 135x24), "Connections: %s", text variable: g_bHMI_EL6900_NoOfConnections
        Label (0,0 135x22), "Safety Project INFO:"
        Rectangle (2,34 135x24), "Groups: %s", text variable: g_bHMI_EL6900_NoOfSafetyGrps
        Rectangle (2,53 135x24), "Safety FBs: %s", text variable: g_bHMI_EL6900_NoOfSafetyFBs
    Button (662,322 110x27), "Error Clear"
        OnMouseUp: execute { g_xHMI_EL6900_ErrClearPB := FALSE ; }
        OnMouseDown: execute { g_xHMI_EL6900_ErrClearPB := TRUE ; }
    Group (168,352 604x31)
        Rectangle (0,0 604x31)
        Label (243,9 118x15), "(3.300 v Nominal)"
        Rectangle (4,5 240x22), "MC1 Actual Voltage: %0.3f v", text variable: g_wHMI_EL6900PriMC_Volts
        Rectangle (362,4 235x22), "MC2 Actual Voltage: %0.3f v", text variable: g_wHMI_EL6900SecMC_Volts
    Group (168,601 603x30)
        Rectangle (0,0 603x30)
        Rectangle (3,4 264x21), "MC1 Actual Temperature: %s C", text variable: g_wHMI_EL6900PriMCTemp
        Rectangle (330,4 270x22), "MC2 Actual Temperature: %s C", text variable: g_wHMI_EL6900SecMCTemp
    Group (168,387 603x210)
        Rectangle (0,0 603x210)
        Label (80,0 130x25), "Temperature Errors"
        Rectangle (6,23 272x32), "Maximum Temperature Exceeded", colour toggle: g_xHMI_EL6900_MaxTemp
        Label (371,0 130x25), "Voltage Errors"
        Rectangle (6,59 272x32), "Temperature Fell Below Minimum", colour toggle: g_xHMI_EL6900_MinTemp
        Rectangle (6,95 272x42), "Temperature Difference Between Measuring Points Exceeded", colour toggle: g_xHMI_EL6900_TempDiffExceeded
        Rectangle (294,23 301x32), "Max Supply Voltage to MC1 Exceeded", colour toggle: g_xHMI_EL6900_MaxVccMC1
        Rectangle (294,59 301x32), "Max Supply Voltage to MC2 Exceeded", colour toggle: g_xHMI_EL6900_MaxVccMC2
        Rectangle (294,95 301x42), "Voltage Fell Below Min Supply Voltage to MC1", colour toggle: g_xHMI_EL6900_MinVccMC1
        Rectangle (294,141 301x42), "Voltage Fell Below Min Supply Voltage to MC2", colour toggle: g_xHMI_EL6900_MinVccMC2
END_VISUALIZATION

// ---- VISUs/EL6930_Specific_Diagnostics.TcVIS
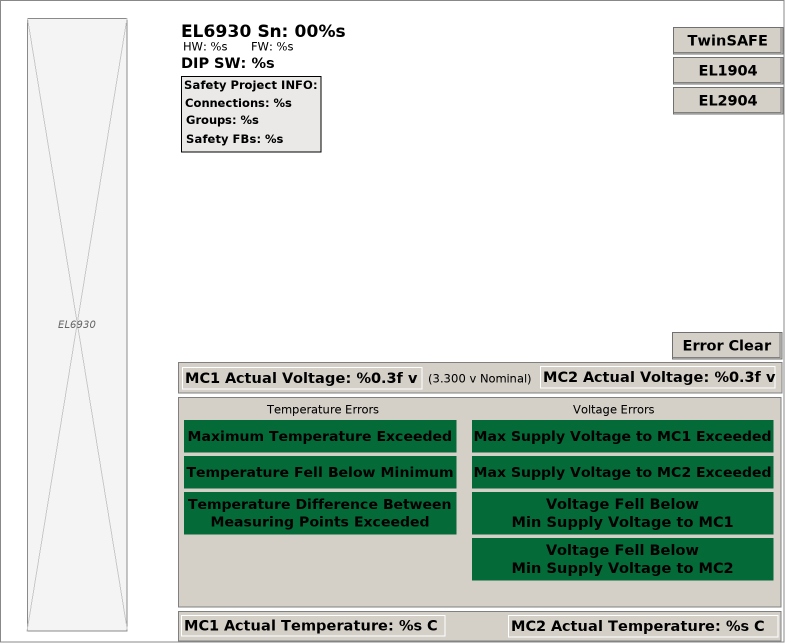
VISUALIZATION EL6930_Specific_Diagnostics  // 785x643
    Button (673,27 110x27), "TwinSAFE"
        OnMouseClick: change screen: TwinSAFE
    Button (673,57 110x27), "EL1904"
        OnMouseClick: change screen: EL1904_Specific_Diagnostics
    Button (673,87 110x27), "EL2904"
        OnMouseClick: change screen: EL2904_Specific_Diagnostics
    Rectangle (178,20 275x22), "EL6930 Sn: 00%s", text variable: g_dwHMI_EL6930Sn
    Rectangle (180,38 65x17), "HW: %s", text variable: g_sHMI_EL6930_HWvers
    Rectangle (248,38 65x17), "FW: %s", text variable: g_sHMI_EL6930_FWvers
    Rectangle (178,52 164x22), "DIP SW: %s", text variable: g_wHMI_EL6930DSw
    Group (181,74 140x78)
        Rectangle (0,2 140x76)
        Rectangle (1,17 135x24), "Connections: %s", text variable: g_bHMI_EL6930_NoOfConnections
        Label (0,0 135x22), "Safety Project INFO:"
        Rectangle (2,34 135x24), "Groups: %s", text variable: g_bHMI_EL6930_NoOfSafetyGrps
        Rectangle (2,53 135x24), "Safety FBs: %s", text variable: g_bHMI_EL6930_NoOfSafetyFBs
    Button (672,332 110x27), "Error Clear"
        OnMouseUp: execute { g_xHMI_EL6930_ErrClearPB := FALSE ; }
        OnMouseDown: execute { g_xHMI_EL6930_ErrClearPB := TRUE ; }
    Group (178,362 604x31)
        Rectangle (0,0 604x31)
        Label (243,9 118x15), "(3.300 v Nominal)"
        Rectangle (4,5 240x22), "MC1 Actual Voltage: %0.3f v", text variable: g_wHMI_EL6930PriMC_Volts
        Rectangle (362,4 235x22), "MC2 Actual Voltage: %0.3f v", text variable: g_wHMI_EL6930SecMC_Volts
    Group (178,611 603x30)
        Rectangle (0,0 603x30)
        Rectangle (3,4 264x21), "MC1 Actual Temperature: %s C", text variable: g_wHMI_EL6930PriMCTemp
        Rectangle (330,4 270x22), "MC2 Actual Temperature: %s C", text variable: g_wHMI_EL6930SecMCTemp
    Group (178,397 603x210)
        Rectangle (0,0 603x210)
        Label (80,0 130x25), "Temperature Errors"
        Rectangle (6,23 272x32), "Maximum Temperature Exceeded", colour toggle: g_xHMI_EL6930_MaxTemp
        Label (371,0 130x25), "Voltage Errors"
        Rectangle (6,59 272x32), "Temperature Fell Below Minimum", colour toggle: g_xHMI_EL6930_MinTemp
        Rectangle (6,95 272x42), "Temperature Difference Between Measuring Points Exceeded", colour toggle: g_xHMI_EL6930_TempDiffExceeded
        Rectangle (294,23 301x32), "Max Supply Voltage to MC1 Exceeded", colour toggle: g_xHMI_EL6930_MaxVccMC1
        Rectangle (294,59 301x32), "Max Supply Voltage to MC2 Exceeded", colour toggle: g_xHMI_EL6930_MaxVccMC2
        Rectangle (294,95 301x42), "Voltage Fell Below Min Supply Voltage to MC1", colour toggle: g_xHMI_EL6930_MinVccMC1
        Rectangle (294,141 301x42), "Voltage Fell Below Min Supply Voltage to MC2", colour toggle: g_xHMI_EL6930_MinVccMC2
    Image (27,18 100x613), image: EL6930
END_VISUALIZATION

// ---- VISUs/EP1908_Specific_Diagnostics.TcVIS
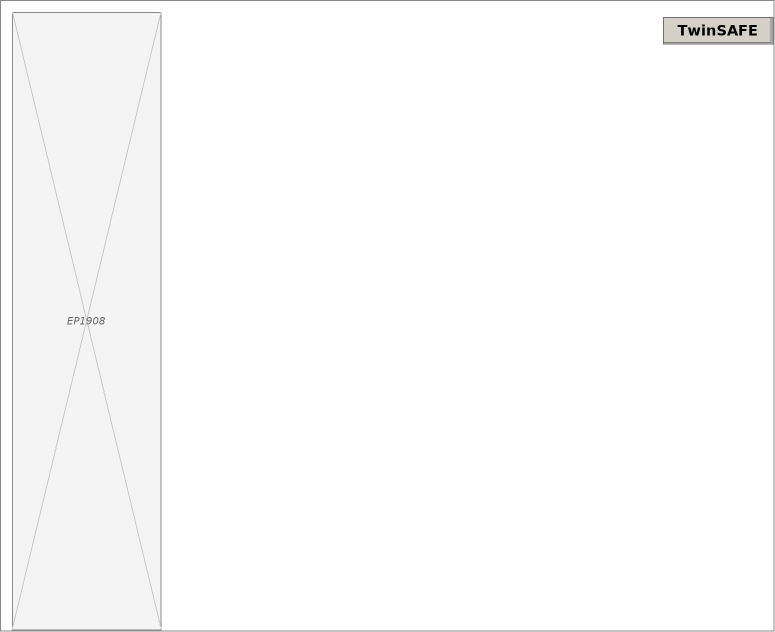
VISUALIZATION EP1908_Specific_Diagnostics  // 775x632
    Button (663,17 110x27), "TwinSAFE"
        OnMouseClick: change screen: TwinSAFE
        OnMouseUp: execute { g_xHMI_ErrAckPB := FALSE ; }
    Image (12,12 149x618), image: EP1908
END_VISUALIZATION

// ---- VISUs/EP1908_Specific_Diagnostics.TcVIS
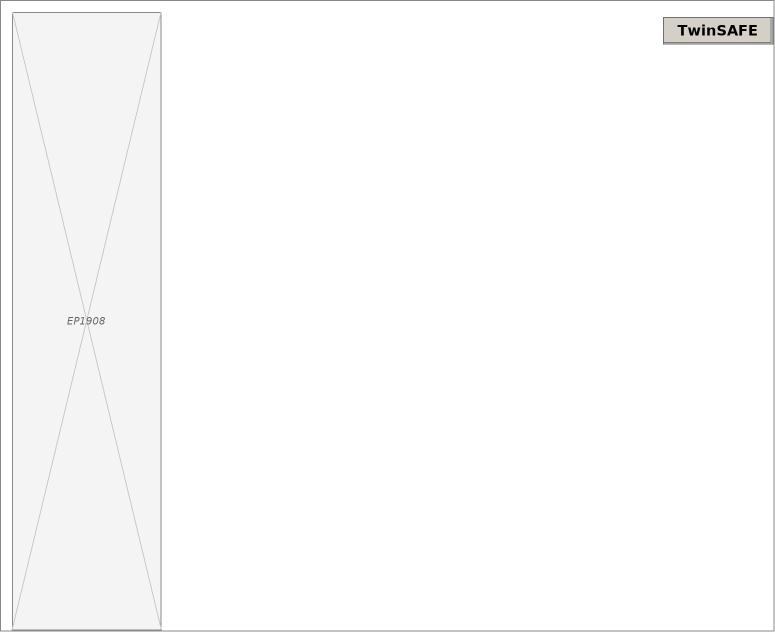
VISUALIZATION EP1908_Specific_Diagnostics  // 775x632
    Button (663,17 110x27), "TwinSAFE"
        OnMouseClick: change screen: TwinSAFE
        OnMouseUp: execute { g_xHMI_ErrAckPB := FALSE ; }
    Image (12,12 149x618), image: EP1908
END_VISUALIZATION

// ---- VISUs/EP1908_Specific_Diagnostics.TcVIS
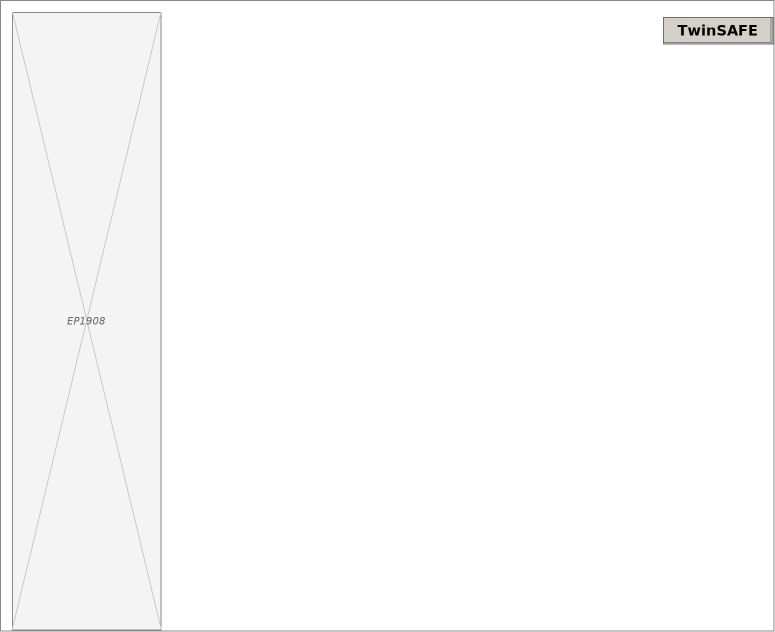
VISUALIZATION EP1908_Specific_Diagnostics  // 775x632
    Button (663,17 110x27), "TwinSAFE"
        OnMouseClick: change screen: TwinSAFE
        OnMouseUp: execute { g_xHMI_ErrAckPB := FALSE ; }
    Image (12,12 149x618), image: EP1908
END_VISUALIZATION

// ---- VISUs/EP1908_Specific_Diagnostics.TcVIS
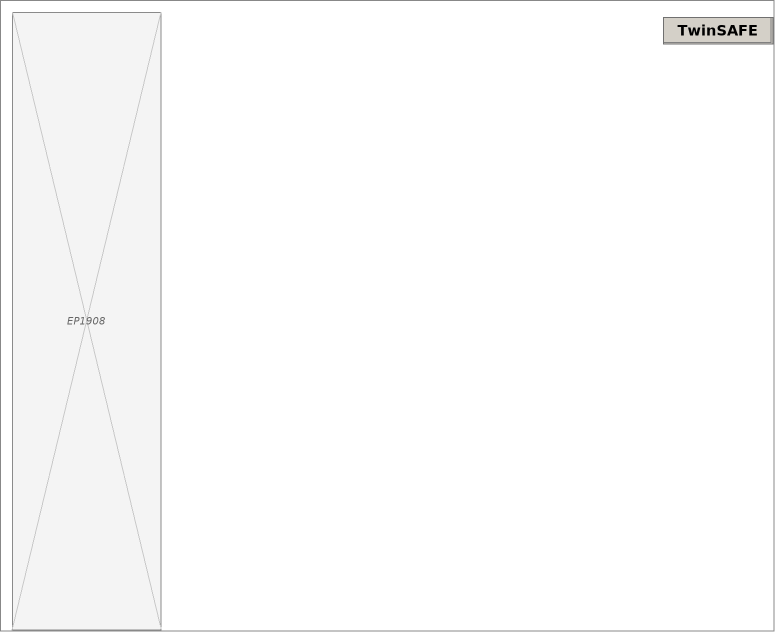
VISUALIZATION EP1908_Specific_Diagnostics  // 775x632
    Button (663,17 110x27), "TwinSAFE"
        OnMouseClick: change screen: TwinSAFE
        OnMouseUp: execute { g_xHMI_ErrAckPB := FALSE ; }
    Image (12,12 149x618), image: EP1908
END_VISUALIZATION

// ---- VISUs/EtherCAT_Diag1.TcVIS
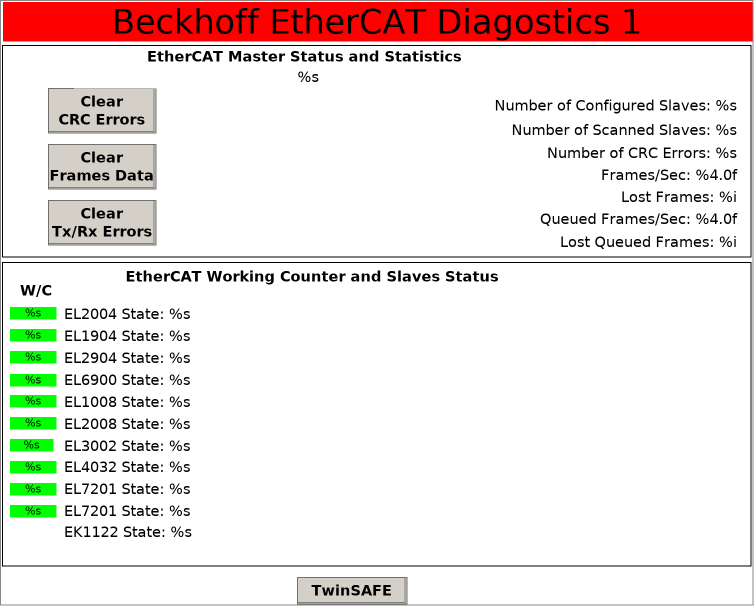
VISUALIZATION EtherCAT_Diag1  // 754x606
    Button (297,577 110x27), "TwinSAFE"
        OnMouseClick: change screen: TwinSAFE
    RoundedRectangle (3,2 749x39), "Beckhoff EtherCAT Diagostics 1"
    RoundedRectangle (2,45 749x212)
    RoundedRectangle (2,262 749x304)
    Label (152,45 305x23), "EtherCAT Master Status and Statistics"
    Button (48,88 108x45), "Clear CRC Errors"
        tap g_xHMI_CearMFStatCRCs
    Label (123,265 378x23), "EtherCAT Working Counter and Slaves Status"
    Button (48,144 108x45), "Clear Frames Data"
        tap g_xHMI_ClearMFStatFrames
    Button (48,200 108x45), "Clear Tx/Rx Errors"
        tap g_xHMI_ClearMFStatTxRxErr
    Label (14,279 44x23), "W/C"
    Rectangle (74,66 469x22), "%s", text variable: g_sHMI_StateMaster
    Rectangle (428,97 312x17), "Number of Configured Slaves: %s", text variable: g_uiHMI_ConfSlaves
    Rectangle (429,121 311x18), "Number of Scanned Slaves: %s", text variable: g_uiHMI_ScannedSlaves
    Rectangle (430,144 310x18), "Number of CRC Errors: %s", text variable: g_dwHMI_TotalCrcErrors
    Rectangle (431,166 309x18), "Frames/Sec: %4.0f", text variable: g_lrHMI_FramesPerSecond
    Rectangle (430,188 310x18), "Lost Frames: %i", text variable: g_udiHMI_LostFrames
    Rectangle (431,210 309x18), "Queued Frames/Sec: %4.0f", text variable: g_lrHMI_QueuedFramesPerSecond
    Rectangle (432,233 308x18), "Lost Queued Frames: %i", text variable: g_udiHMI_LostQueuedFrames
    Rectangle (61,303 686x22), "EL2004 State: %s", text variable: g_sHMI_StateEL2004
    Rectangle (61,325 685x22), "EL1904 State: %s", text variable: g_sHMI_StateEL1904
    Rectangle (61,347 686x22), "EL2904 State: %s", text variable: g_sHMI_StateEL2904
    Rectangle (61,369 684x22), "EL6900 State: %s", text variable: g_sHMI_StateEL6900
    Rectangle (61,391 683x22), "EL1008 State: %s", text variable: g_sHMI_StateEL1008
    Rectangle (61,413 685x22), "EL2008 State: %s", text variable: g_sHMI_StateEL2008
    Rectangle (61,435 685x22), "EL3002 State: %s", text variable: g_sHMI_StateEL3002
    Rectangle (61,456 684x22), "EL4032 State: %s", text variable: g_sHMI_StateEL4032
    Rectangle (10,307 46x12), "%s", text variable: g_xEL2004_Wc
    Rectangle (10,329 46x12), "%s", text variable: g_xEL1904_Wc
    Rectangle (10,351 46x12), "%s", text variable: g_xEL2904_Wc
    Rectangle (10,374 46x12), "%s", text variable: g_xEL6900_Wc
    Rectangle (10,395 46x12), "%s", text variable: g_xEL1008_Wc
    Rectangle (10,417 46x12), "%s", text variable: g_xEL2008_Wc
    Rectangle (10,439 43x12), "%s", text variable: g_xEL3002_Wc
    Rectangle (10,461 46x12), "%s", text variable: g_xEL4032_Wc
    Rectangle (61,478 684x22), "EL7201 State: %s", text variable: g_sHMI_StateEL7201_1
    Rectangle (10,483 46x12), "%s", text variable: g_xEL7201_2_Wc
    Rectangle (61,500 684x22), "EL7201 State: %s", text variable: g_sHMI_StateEL7201_2
    Rectangle (10,505 46x12), "%s", text variable: g_xEL7201_2_Wc
    Rectangle (61,521 684x22), "EK1122 State: %s", text variable: g_sHMI_StateEK1122
END_VISUALIZATION

// ---- VISUs/EtherCAT_Diag1.TcVIS
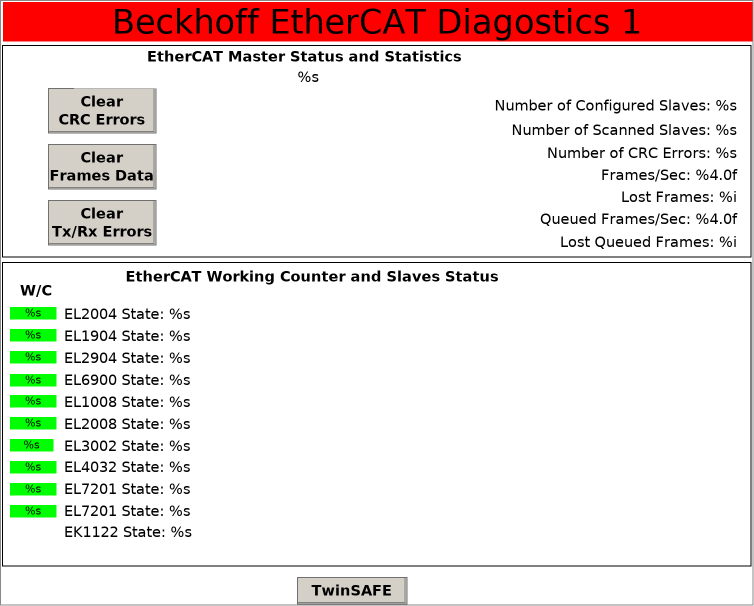
VISUALIZATION EtherCAT_Diag1  // 754x606
    Button (297,577 110x27), "TwinSAFE"
        OnMouseClick: change screen: TwinSAFE
    RoundedRectangle (3,2 749x39), "Beckhoff EtherCAT Diagostics 1"
    RoundedRectangle (2,45 749x212)
    RoundedRectangle (2,262 749x304)
    Label (152,45 305x23), "EtherCAT Master Status and Statistics"
    Button (48,88 108x45), "Clear CRC Errors"
        tap g_xHMI_CearMFStatCRCs
    Label (123,265 378x23), "EtherCAT Working Counter and Slaves Status"
    Button (48,144 108x45), "Clear Frames Data"
        tap g_xHMI_ClearMFStatFrames
    Button (48,200 108x45), "Clear Tx/Rx Errors"
        tap g_xHMI_ClearMFStatTxRxErr
    Label (14,279 44x23), "W/C"
    Rectangle (74,66 469x22), "%s", text variable: g_sHMI_StateMaster
    Rectangle (428,97 312x17), "Number of Configured Slaves: %s", text variable: g_uiHMI_ConfSlaves
    Rectangle (429,121 311x18), "Number of Scanned Slaves: %s", text variable: g_uiHMI_ScannedSlaves
    Rectangle (430,144 310x18), "Number of CRC Errors: %s", text variable: g_dwHMI_TotalCrcErrors
    Rectangle (431,166 309x18), "Frames/Sec: %4.0f", text variable: g_lrHMI_FramesPerSecond
    Rectangle (430,188 310x18), "Lost Frames: %i", text variable: g_udiHMI_LostFrames
    Rectangle (431,210 309x18), "Queued Frames/Sec: %4.0f", text variable: g_lrHMI_QueuedFramesPerSecond
    Rectangle (432,233 308x18), "Lost Queued Frames: %i", text variable: g_udiHMI_LostQueuedFrames
    Rectangle (61,303 686x22), "EL2004 State: %s", text variable: g_sHMI_StateEL2004
    Rectangle (61,325 685x22), "EL1904 State: %s", text variable: g_sHMI_StateEL1904
    Rectangle (61,347 686x22), "EL2904 State: %s", text variable: g_sHMI_StateEL2904
    Rectangle (61,369 684x22), "EL6900 State: %s", text variable: g_sHMI_StateEL6900
    Rectangle (61,391 683x22), "EL1008 State: %s", text variable: g_sHMI_StateEL1008
    Rectangle (61,413 685x22), "EL2008 State: %s", text variable: g_sHMI_StateEL2008
    Rectangle (61,435 685x22), "EL3002 State: %s", text variable: g_sHMI_StateEL3002
    Rectangle (61,456 684x22), "EL4032 State: %s", text variable: g_sHMI_StateEL4032
    Rectangle (10,307 46x12), "%s", text variable: g_xEL2004_Wc
    Rectangle (10,329 46x12), "%s", text variable: g_xEL1904_Wc
    Rectangle (10,351 46x12), "%s", text variable: g_xEL2904_Wc
    Rectangle (10,374 46x12), "%s", text variable: g_xEL6900_Wc
    Rectangle (10,395 46x12), "%s", text variable: g_xEL1008_Wc
    Rectangle (10,417 46x12), "%s", text variable: g_xEL2008_Wc
    Rectangle (10,439 43x12), "%s", text variable: g_xEL3002_Wc
    Rectangle (10,461 46x12), "%s", text variable: g_xEL4032_Wc
    Rectangle (61,478 684x22), "EL7201 State: %s", text variable: g_sHMI_StateEL7201_1
    Rectangle (10,483 46x12), "%s", text variable: g_xEL7201_2_Wc
    Rectangle (61,500 684x22), "EL7201 State: %s", text variable: g_sHMI_StateEL7201_2
    Rectangle (10,505 46x12), "%s", text variable: g_xEL7201_2_Wc
    Rectangle (61,521 684x22), "EK1122 State: %s", text variable: g_sHMI_StateEK1122
END_VISUALIZATION

// ---- VISUs/EtherCAT_Diag1.TcVIS
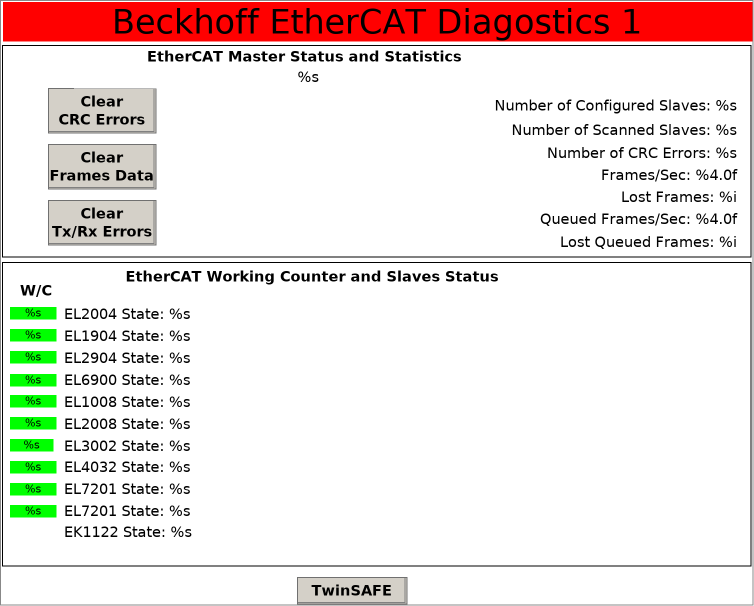
VISUALIZATION EtherCAT_Diag1  // 754x606
    Button (297,577 110x27), "TwinSAFE"
        OnMouseClick: change screen: TwinSAFE
    RoundedRectangle (3,2 749x39), "Beckhoff EtherCAT Diagostics 1"
    RoundedRectangle (2,45 749x212)
    RoundedRectangle (2,262 749x304)
    Label (152,45 305x23), "EtherCAT Master Status and Statistics"
    Button (48,88 108x45), "Clear CRC Errors"
        tap g_xHMI_CearMFStatCRCs
    Label (123,265 378x23), "EtherCAT Working Counter and Slaves Status"
    Button (48,144 108x45), "Clear Frames Data"
        tap g_xHMI_ClearMFStatFrames
    Button (48,200 108x45), "Clear Tx/Rx Errors"
        tap g_xHMI_ClearMFStatTxRxErr
    Label (14,279 44x23), "W/C"
    Rectangle (74,66 469x22), "%s", text variable: g_sHMI_StateMaster
    Rectangle (428,97 312x17), "Number of Configured Slaves: %s", text variable: g_uiHMI_ConfSlaves
    Rectangle (429,121 311x18), "Number of Scanned Slaves: %s", text variable: g_uiHMI_ScannedSlaves
    Rectangle (430,144 310x18), "Number of CRC Errors: %s", text variable: g_dwHMI_TotalCrcErrors
    Rectangle (431,166 309x18), "Frames/Sec: %4.0f", text variable: g_lrHMI_FramesPerSecond
    Rectangle (430,188 310x18), "Lost Frames: %i", text variable: g_udiHMI_LostFrames
    Rectangle (431,210 309x18), "Queued Frames/Sec: %4.0f", text variable: g_lrHMI_QueuedFramesPerSecond
    Rectangle (432,233 308x18), "Lost Queued Frames: %i", text variable: g_udiHMI_LostQueuedFrames
    Rectangle (61,303 686x22), "EL2004 State: %s", text variable: g_sHMI_StateEL2004
    Rectangle (61,325 685x22), "EL1904 State: %s", text variable: g_sHMI_StateEL1904
    Rectangle (61,347 686x22), "EL2904 State: %s", text variable: g_sHMI_StateEL2904
    Rectangle (61,369 684x22), "EL6900 State: %s", text variable: g_sHMI_StateEL6900
    Rectangle (61,391 683x22), "EL1008 State: %s", text variable: g_sHMI_StateEL1008
    Rectangle (61,413 685x22), "EL2008 State: %s", text variable: g_sHMI_StateEL2008
    Rectangle (61,435 685x22), "EL3002 State: %s", text variable: g_sHMI_StateEL3002
    Rectangle (61,456 684x22), "EL4032 State: %s", text variable: g_sHMI_StateEL4032
    Rectangle (10,307 46x12), "%s", text variable: g_xEL2004_Wc
    Rectangle (10,329 46x12), "%s", text variable: g_xEL1904_Wc
    Rectangle (10,351 46x12), "%s", text variable: g_xEL2904_Wc
    Rectangle (10,374 46x12), "%s", text variable: g_xEL6900_Wc
    Rectangle (10,395 46x12), "%s", text variable: g_xEL1008_Wc
    Rectangle (10,417 46x12), "%s", text variable: g_xEL2008_Wc
    Rectangle (10,439 43x12), "%s", text variable: g_xEL3002_Wc
    Rectangle (10,461 46x12), "%s", text variable: g_xEL4032_Wc
    Rectangle (61,478 684x22), "EL7201 State: %s", text variable: g_sHMI_StateEL7201_1
    Rectangle (10,483 46x12), "%s", text variable: g_xEL7201_2_Wc
    Rectangle (61,500 684x22), "EL7201 State: %s", text variable: g_sHMI_StateEL7201_2
    Rectangle (10,505 46x12), "%s", text variable: g_xEL7201_2_Wc
    Rectangle (61,521 684x22), "EK1122 State: %s", text variable: g_sHMI_StateEK1122
END_VISUALIZATION

// ---- VISUs/EtherCAT_Diag2.TcVIS
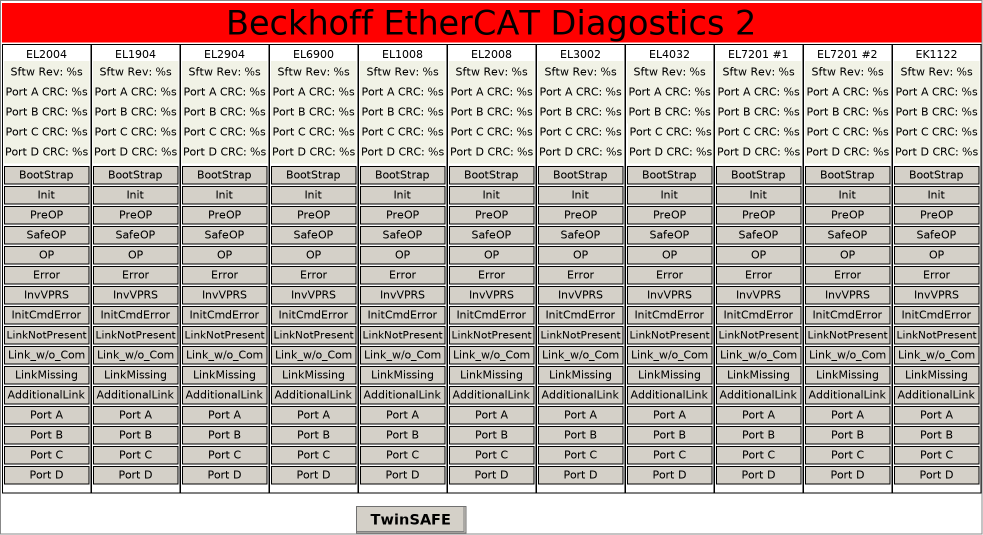
VISUALIZATION EtherCAT_Diag2  // 983x535
    Button (356,506 110x27), "TwinSAFE"
        OnMouseClick: change screen: TwinSAFE
    RoundedRectangle (2,3 979x39), "Beckhoff EtherCAT Diagostics 2"
    Group (2,42 89x451)
        RoundedRectangle (0,2 89x449)
        Label (2,0 85x25), "EL2004"
        Rectangle (2,19 85x22), "Sftw Rev: %s", text variable: g_iHMI_ProdCodeEL2004
        Rectangle (2,39 85x22), "Port A CRC: %s", text variable: g_stHMI_EL2004CrcErrorEx.portA
        Rectangle (2,59 85x22), "Port B CRC: %s", text variable: g_stHMI_EL2004CrcErrorEx.portB
        Rectangle (2,79 85x22), "Port C CRC: %s", text variable: g_stHMI_EL2004CrcErrorEx.portC
        Rectangle (2,99 85x22), "Port D CRC: %s", text variable: g_stHMI_EL2004CrcErrorEx.portD
        Rectangle (2,124 85x18), "BootStrap", colour toggle: g_stHMI_EL2004EcSlaveStateBits.bBootStrap
        Rectangle (2,144 85x18), "Init", colour toggle: g_stHMI_EL2004EcSlaveStateBits.bInit
        Rectangle (2,164 85x18), "PreOP", colour toggle: g_stHMI_EL2004EcSlaveStateBits.bPreop
        Rectangle (2,184 85x18), "SafeOP", colour toggle: g_stHMI_EL2004EcSlaveStateBits.bSafeOp
        Rectangle (2,204 85x18), "OP", colour toggle: g_stHMI_EL2004EcSlaveStateBits.bOp
        Rectangle (2,224 85x18), "Error", colour toggle: g_stHMI_EL2004EcSlaveStateBits.bError
        Rectangle (2,244 85x18), "InvVPRS", colour toggle: g_stHMI_EL2004EcSlaveStateBits.bInvVPRS
        Rectangle (2,264 85x18), "InitCmdError", colour toggle: g_stHMI_EL2004EcSlaveStateBits.bInitCmdError
        Rectangle (2,284 85x18), "LinkNotPresent", colour toggle: g_stHMI_EL2004EcSlaveStateBits.bLinkNotPresent
        Rectangle (2,304 85x18), "Link_w/o_Com", colour toggle: g_stHMI_EL2004EcSlaveStateBits.bLinkWithoutComm
        Rectangle (2,324 85x18), "LinkMissing", colour toggle: g_stHMI_EL2004EcSlaveStateBits.bLinkMissing
        Rectangle (2,344 85x18), "AdditionalLink", colour toggle: g_stHMI_EL2004EcSlaveStateBits.bAdditionalLink
        Rectangle (2,364 85x18), "Port A", colour toggle: g_stHMI_EL2004EcSlaveStateBits.bPortA
        Rectangle (2,384 85x18), "Port B", colour toggle: g_stHMI_EL2004EcSlaveStateBits.bPortB
        Rectangle (2,404 85x18), "Port C", colour toggle: g_stHMI_EL2004EcSlaveStateBits.bPortC
        Rectangle (2,424 85x18), "Port D", colour toggle: g_stHMI_EL2004EcSlaveStateBits.bPortD
    Group (91,42 89x451)
        RoundedRectangle (0,2 89x449)
        Label (2,0 85x25), "EL1904"
        Rectangle (2,19 85x22), "Sftw Rev: %s", text variable: g_iHMI_ProdCodeEL1904
        Rectangle (2,39 85x22), "Port A CRC: %s", text variable: g_stHMI_EL1904CrcErrorEx.portA
        Rectangle (2,59 85x22), "Port B CRC: %s", text variable: g_stHMI_EL1904CrcErrorEx.portB
        Rectangle (2,79 85x22), "Port C CRC: %s", text variable: g_stHMI_EL1904CrcErrorEx.portC
        Rectangle (2,99 85x22), "Port D CRC: %s", text variable: g_stHMI_EL1904CrcErrorEx.portD
        Rectangle (2,124 85x18), "BootStrap", colour toggle: g_stHMI_EL1904EcSlaveStateBits.bBootStrap
        Rectangle (2,144 85x18), "Init", colour toggle: g_stHMI_EL1904EcSlaveStateBits.bInit
        Rectangle (2,164 85x18), "PreOP", colour toggle: g_stHMI_EL1904EcSlaveStateBits.bPreop
        Rectangle (2,184 85x18), "SafeOP", colour toggle: g_stHMI_EL1904EcSlaveStateBits.bSafeOp
        Rectangle (2,204 85x18), "OP", colour toggle: g_stHMI_EL1904EcSlaveStateBits.bOp
        Rectangle (2,224 85x18), "Error", colour toggle: g_stHMI_EL1904EcSlaveStateBits.bError
        Rectangle (2,244 85x18), "InvVPRS", colour toggle: g_stHMI_EL1904EcSlaveStateBits.bInvVPRS
        Rectangle (2,264 85x18), "InitCmdError", colour toggle: g_stHMI_EL1904EcSlaveStateBits.bInitCmdError
        Rectangle (2,284 85x18), "LinkNotPresent", colour toggle: g_stHMI_EL1904EcSlaveStateBits.bLinkNotPresent
        Rectangle (2,304 85x18), "Link_w/o_Com", colour toggle: g_stHMI_EL1904EcSlaveStateBits.bLinkWithoutComm
        Rectangle (2,324 85x18), "LinkMissing", colour toggle: g_stHMI_EL1904EcSlaveStateBits.bLinkMissing
        Rectangle (2,344 85x18), "AdditionalLink", colour toggle: g_stHMI_EL1904EcSlaveStateBits.bAdditionalLink
        Rectangle (2,364 85x18), "Port A", colour toggle: g_stHMI_EL1904EcSlaveStateBits.bPortA
        Rectangle (2,384 85x18), "Port B", colour toggle: g_stHMI_EL1904EcSlaveStateBits.bPortB
        Rectangle (2,404 85x18), "Port C", colour toggle: g_stHMI_EL1904EcSlaveStateBits.bPortC
        Rectangle (2,424 85x18), "Port D", colour toggle: g_stHMI_EL1904EcSlaveStateBits.bPortD
    Group (180,42 89x451)
        RoundedRectangle (0,2 89x449)
        Label (2,0 85x25), "EL2904"
        Rectangle (2,19 85x22), "Sftw Rev: %s", text variable: g_iHMI_ProdCodeEL2904
        Rectangle (2,39 85x22), "Port A CRC: %s", text variable: g_stHMI_EL2904CrcErrorEx.portA
        Rectangle (2,59 85x22), "Port B CRC: %s", text variable: g_stHMI_EL2904CrcErrorEx.portB
        Rectangle (2,79 85x22), "Port C CRC: %s", text variable: g_stHMI_EL2904CrcErrorEx.portC
        Rectangle (2,99 85x22), "Port D CRC: %s", text variable: g_stHMI_EL2904CrcErrorEx.portD
        Rectangle (2,124 85x18), "BootStrap", colour toggle: g_stHMI_EL2904EcSlaveStateBits.bBootStrap
        Rectangle (2,144 85x18), "Init", colour toggle: g_stHMI_EL2904EcSlaveStateBits.bInit
        Rectangle (2,164 85x18), "PreOP", colour toggle: g_stHMI_EL2904EcSlaveStateBits.bPreop
        Rectangle (2,184 85x18), "SafeOP", colour toggle: g_stHMI_EL2904EcSlaveStateBits.bSafeOp
        Rectangle (2,204 85x18), "OP", colour toggle: g_stHMI_EL2904EcSlaveStateBits.bOp
        Rectangle (2,224 85x18), "Error", colour toggle: g_stHMI_EL2904EcSlaveStateBits.bError
        Rectangle (2,244 85x18), "InvVPRS", colour toggle: g_stHMI_EL2904EcSlaveStateBits.bInvVPRS
        Rectangle (2,264 85x18), "InitCmdError", colour toggle: g_stHMI_EL2904EcSlaveStateBits.bInitCmdError
        Rectangle (2,284 85x18), "LinkNotPresent", colour toggle: g_stHMI_EL2904EcSlaveStateBits.bLinkNotPresent
        Rectangle (2,304 85x18), "Link_w/o_Com", colour toggle: g_stHMI_EL2904EcSlaveStateBits.bLinkWithoutComm
        Rectangle (2,324 85x18), "LinkMissing", colour toggle: g_stHMI_EL2904EcSlaveStateBits.bLinkMissing
        Rectangle (2,344 85x18), "AdditionalLink", colour toggle: g_stHMI_EL2904EcSlaveStateBits.bAdditionalLink
        Rectangle (2,364 85x18), "Port A", colour toggle: g_stHMI_EL2904EcSlaveStateBits.bPortA
        Rectangle (2,384 85x18), "Port B", colour toggle: g_stHMI_EL2904EcSlaveStateBits.bPortB
        Rectangle (2,404 85x18), "Port C", colour toggle: g_stHMI_EL2904EcSlaveStateBits.bPortC
        Rectangle (2,424 85x18), "Port D", colour toggle: g_stHMI_EL2904EcSlaveStateBits.bPortD
    Group (269,42 89x451)
        RoundedRectangle (0,2 89x449)
        Label (2,0 85x25), "EL6900"
        Rectangle (2,19 85x22), "Sftw Rev: %s", text variable: g_iHMI_ProdCodeEL6900
        Rectangle (2,39 85x22), "Port A CRC: %s", text variable: g_stHMI_EL6900CrcErrorEx.portA
        Rectangle (2,59 85x22), "Port B CRC: %s", text variable: g_stHMI_EL6900CrcErrorEx.portB
        Rectangle (2,79 85x22), "Port C CRC: %s", text variable: g_stHMI_EL6900CrcErrorEx.portC
        Rectangle (2,99 85x22), "Port D CRC: %s", text variable: g_stHMI_EL6900CrcErrorEx.portD
        Rectangle (2,124 85x18), "BootStrap", colour toggle: g_stHMI_EL6900EcSlaveStateBits.bBootStrap
        Rectangle (2,144 85x18), "Init", colour toggle: g_stHMI_EL6900EcSlaveStateBits.bInit
        Rectangle (2,164 85x18), "PreOP", colour toggle: g_stHMI_EL6900EcSlaveStateBits.bPreop
        Rectangle (2,184 85x18), "SafeOP", colour toggle: g_stHMI_EL6900EcSlaveStateBits.bSafeOp
        Rectangle (2,204 85x18), "OP", colour toggle: g_stHMI_EL6900EcSlaveStateBits.bOp
        Rectangle (2,224 85x18), "Error", colour toggle: g_stHMI_EL6900EcSlaveStateBits.bError
        Rectangle (2,244 85x18), "InvVPRS", colour toggle: g_stHMI_EL6900EcSlaveStateBits.bInvVPRS
        Rectangle (2,264 85x18), "InitCmdError", colour toggle: g_stHMI_EL6900EcSlaveStateBits.bInitCmdError
        Rectangle (2,284 85x18), "LinkNotPresent", colour toggle: g_stHMI_EL6900EcSlaveStateBits.bLinkNotPresent
        Rectangle (2,304 85x18), "Link_w/o_Com", colour toggle: g_stHMI_EL6900EcSlaveStateBits.bLinkWithoutComm
        Rectangle (2,324 85x18), "LinkMissing", colour toggle: g_stHMI_EL6900EcSlaveStateBits.bLinkMissing
        Rectangle (2,344 85x18), "AdditionalLink", colour toggle: g_stHMI_EL6900EcSlaveStateBits.bAdditionalLink
        Rectangle (2,364 85x18), "Port A", colour toggle: g_stHMI_EL6900EcSlaveStateBits.bPortA
        Rectangle (2,384 85x18), "Port B", colour toggle: g_stHMI_EL6900EcSlaveStateBits.bPortB
        Rectangle (2,404 85x18), "Port C", colour toggle: g_stHMI_EL6900EcSlaveStateBits.bPortC
        Rectangle (2,424 85x18), "Port D", colour toggle: g_stHMI_EL6900EcSlaveStateBits.bPortD
    Group (358,42 89x451)
        RoundedRectangle (0,2 89x449)
        Label (2,0 85x25), "EL1008"
        Rectangle (2,19 85x22), "Sftw Rev: %s", text variable: g_iHMI_ProdCodeEL1008
        Rectangle (2,39 85x22), "Port A CRC: %s", text variable: g_stHMI_EL1008CrcErrorEx.portA
        Rectangle (2,59 85x22), "Port B CRC: %s", text variable: g_stHMI_EL1008CrcErrorEx.portB
        Rectangle (2,79 85x22), "Port C CRC: %s", text variable: g_stHMI_EL1008CrcErrorEx.portC
        Rectangle (2,99 85x22), "Port D CRC: %s", text variable: g_stHMI_EL1008CrcErrorEx.portD
        Rectangle (2,124 85x18), "BootStrap", colour toggle: g_stHMI_EL1008EcSlaveStateBits.bBootStrap
        Rectangle (2,144 85x18), "Init", colour toggle: g_stHMI_EL1008EcSlaveStateBits.bInit
        Rectangle (2,164 85x18), "PreOP", colour toggle: g_stHMI_EL1008EcSlaveStateBits.bPreop
        Rectangle (2,184 85x18), "SafeOP", colour toggle: g_stHMI_EL1008EcSlaveStateBits.bSafeOp
        Rectangle (2,204 85x18), "OP", colour toggle: g_stHMI_EL1008EcSlaveStateBits.bOp
        Rectangle (2,224 85x18), "Error", colour toggle: g_stHMI_EL1008EcSlaveStateBits.bError
        Rectangle (2,244 85x18), "InvVPRS", colour toggle: g_stHMI_EL1008EcSlaveStateBits.bInvVPRS
        Rectangle (2,264 85x18), "InitCmdError", colour toggle: g_stHMI_EL1008EcSlaveStateBits.bInitCmdError
        Rectangle (2,284 85x18), "LinkNotPresent", colour toggle: g_stHMI_EL1008EcSlaveStateBits.bLinkNotPresent
        Rectangle (2,304 85x18), "Link_w/o_Com", colour toggle: g_stHMI_EL1008EcSlaveStateBits.bLinkWithoutComm
        Rectangle (2,324 85x18), "LinkMissing", colour toggle: g_stHMI_EL1008EcSlaveStateBits.bLinkMissing
        Rectangle (2,344 85x18), "AdditionalLink", colour toggle: g_stHMI_EL1008EcSlaveStateBits.bAdditionalLink
        Rectangle (2,364 85x18), "Port A", colour toggle: g_stHMI_EL1008EcSlaveStateBits.bPortA
        Rectangle (2,384 85x18), "Port B", colour toggle: g_stHMI_EL1008EcSlaveStateBits.bPortB
        Rectangle (2,404 85x18), "Port C", colour toggle: g_stHMI_EL1008EcSlaveStateBits.bPortC
        Rectangle (2,424 85x18), "Port D", colour toggle: g_stHMI_EL1008EcSlaveStateBits.bPortD
    Group (447,42 89x451)
        RoundedRectangle (0,2 89x449)
        Label (2,0 85x25), "EL2008"
        Rectangle (2,19 85x22), "Sftw Rev: %s", text variable: g_iHMI_ProdCodeEL2008
        Rectangle (2,39 85x22), "Port A CRC: %s", text variable: g_stHMI_EL2008CrcErrorEx.portA
        Rectangle (2,59 85x22), "Port B CRC: %s", text variable: g_stHMI_EL2008CrcErrorEx.portB
        Rectangle (2,79 85x22), "Port C CRC: %s", text variable: g_stHMI_EL2008CrcErrorEx.portC
        Rectangle (2,99 85x22), "Port D CRC: %s", text variable: g_stHMI_EL2008CrcErrorEx.portD
        Rectangle (2,124 85x18), "BootStrap", colour toggle: g_stHMI_EL2008EcSlaveStateBits.bBootStrap
        Rectangle (2,144 85x18), "Init", colour toggle: g_stHMI_EL2008EcSlaveStateBits.bInit
        Rectangle (2,164 85x18), "PreOP", colour toggle: g_stHMI_EL2008EcSlaveStateBits.bPreop
        Rectangle (2,184 85x18), "SafeOP", colour toggle: g_stHMI_EL2008EcSlaveStateBits.bSafeOp
        Rectangle (2,204 85x18), "OP", colour toggle: g_stHMI_EL2008EcSlaveStateBits.bOp
        Rectangle (2,224 85x18), "Error", colour toggle: g_stHMI_EL2008EcSlaveStateBits.bError
        Rectangle (2,244 85x18), "InvVPRS", colour toggle: g_stHMI_EL2008EcSlaveStateBits.bInvVPRS
        Rectangle (2,264 85x18), "InitCmdError", colour toggle: g_stHMI_EL2008EcSlaveStateBits.bInitCmdError
        Rectangle (2,284 85x18), "LinkNotPresent", colour toggle: g_stHMI_EL2008EcSlaveStateBits.bLinkNotPresent
        Rectangle (2,304 85x18), "Link_w/o_Com", colour toggle: g_stHMI_EL2008EcSlaveStateBits.bLinkWithoutComm
        Rectangle (2,324 85x18), "LinkMissing", colour toggle: g_stHMI_EL2008EcSlaveStateBits.bLinkMissing
        Rectangle (2,344 85x18), "AdditionalLink", colour toggle: g_stHMI_EL2008EcSlaveStateBits.bAdditionalLink
        Rectangle (2,364 85x18), "Port A", colour toggle: g_stHMI_EL2008EcSlaveStateBits.bPortA
        Rectangle (2,384 85x18), "Port B", colour toggle: g_stHMI_EL2008EcSlaveStateBits.bPortB
        Rectangle (2,404 85x18), "Port C", colour toggle: g_stHMI_EL2008EcSlaveStateBits.bPortC
        Rectangle (2,424 85x18), "Port D", colour toggle: g_stHMI_EL2008EcSlaveStateBits.bPortD
    Group (536,42 89x451)
        RoundedRectangle (0,2 89x449)
        Label (2,0 85x25), "EL3002"
        Rectangle (2,19 85x22), "Sftw Rev: %s", text variable: g_iHMI_ProdCodeEL3002
        Rectangle (2,39 85x22), "Port A CRC: %s", text variable: g_stHMI_EL3002CrcErrorEx.portA
        Rectangle (2,59 85x22), "Port B CRC: %s", text variable: g_stHMI_EL3002CrcErrorEx.portB
        Rectangle (2,79 85x22), "Port C CRC: %s", text variable: g_stHMI_EL3002CrcErrorEx.portC
        Rectangle (2,99 85x22), "Port D CRC: %s", text variable: g_stHMI_EL3002CrcErrorEx.portD
        Rectangle (2,124 85x18), "BootStrap", colour toggle: g_stHMI_EL3002EcSlaveStateBits.bBootStrap
        Rectangle (2,144 85x18), "Init", colour toggle: g_stHMI_EL3002EcSlaveStateBits.bInit
        Rectangle (2,164 85x18), "PreOP", colour toggle: g_stHMI_EL3002EcSlaveStateBits.bPreop
        Rectangle (2,184 85x18), "SafeOP", colour toggle: g_stHMI_EL3002EcSlaveStateBits.bSafeOp
        Rectangle (2,204 85x18), "OP", colour toggle: g_stHMI_EL3002EcSlaveStateBits.bOp
        Rectangle (2,224 85x18), "Error", colour toggle: g_stHMI_EL3002EcSlaveStateBits.bError
        Rectangle (2,244 85x18), "InvVPRS", colour toggle: g_stHMI_EL3002EcSlaveStateBits.bInvVPRS
        Rectangle (2,264 85x18), "InitCmdError", colour toggle: g_stHMI_EL3002EcSlaveStateBits.bInitCmdError
        Rectangle (2,284 85x18), "LinkNotPresent", colour toggle: g_stHMI_EL3002EcSlaveStateBits.bLinkNotPresent
        Rectangle (2,304 85x18), "Link_w/o_Com", colour toggle: g_stHMI_EL3002EcSlaveStateBits.bLinkWithoutComm
        Rectangle (2,324 85x18), "LinkMissing", colour toggle: g_stHMI_EL3002EcSlaveStateBits.bLinkMissing
        Rectangle (2,344 85x18), "AdditionalLink", colour toggle: g_stHMI_EL3002EcSlaveStateBits.bAdditionalLink
        Rectangle (2,364 85x18), "Port A", colour toggle: g_stHMI_EL3002EcSlaveStateBits.bPortA
        Rectangle (2,384 85x18), "Port B", colour toggle: g_stHMI_EL3002EcSlaveStateBits.bPortB
        Rectangle (2,404 85x18), "Port C", colour toggle: g_stHMI_EL3002EcSlaveStateBits.bPortC
        Rectangle (2,424 85x18), "Port D", colour toggle: g_stHMI_EL3002EcSlaveStateBits.bPortD
    RoundedRectangle (625,44 89x449)
    Label (627,42 85x25), "EL4032"
    Rectangle (627,61 85x22), "Sftw Rev: %s", text variable: g_iHMI_ProdCodeEL4032
    Rectangle (627,81 85x22), "Port A CRC: %s", text variable: g_stHMI_EL4032CrcErrorEx.portA
    Rectangle (627,101 85x22), "Port B CRC: %s", text variable: g_stHMI_EL4032CrcErrorEx.portB
    Rectangle (628,121 85x22), "Port C CRC: %s", text variable: g_stHMI_EL4032CrcErrorEx.portC
    Rectangle (628,141 85x22), "Port D CRC: %s", text variable: g_stHMI_EL4032CrcErrorEx.portD
    Rectangle (627,166 85x18), "BootStrap", colour toggle: g_stHMI_EL4032EcSlaveStateBits.bBootStrap
    Rectangle (627,186 85x18), "Init", colour toggle: g_stHMI_EL4032EcSlaveStateBits.bInit
    Rectangle (627,206 85x18), "PreOP", colour toggle: g_stHMI_EL4032EcSlaveStateBits.bPreop
    Rectangle (627,226 85x18), "SafeOP", colour toggle: g_stHMI_EL4032EcSlaveStateBits.bSafeOp
    Rectangle (627,246 85x18), "OP", colour toggle: g_stHMI_EL4032EcSlaveStateBits.bOp
    Rectangle (627,266 85x18), "Error", colour toggle: g_stHMI_EL4032EcSlaveStateBits.bError
    Rectangle (627,286 85x18), "InvVPRS", colour toggle: g_stHMI_EL4032EcSlaveStateBits.bInvVPRS
    Rectangle (627,306 85x18), "InitCmdError", colour toggle: g_stHMI_EL4032EcSlaveStateBits.bInitCmdError
    Rectangle (627,326 85x18), "LinkNotPresent", colour toggle: g_stHMI_EL4032EcSlaveStateBits.bLinkNotPresent
    Rectangle (627,346 85x18), "Link_w/o_Com", colour toggle: g_stHMI_EL4032EcSlaveStateBits.bLinkWithoutComm
    Rectangle (627,366 85x18), "LinkMissing", colour toggle: g_stHMI_EL4032EcSlaveStateBits.bLinkMissing
    Rectangle (627,386 85x18), "AdditionalLink", colour toggle: g_stHMI_EL4032EcSlaveStateBits.bAdditionalLink
    Rectangle (627,406 85x18), "Port A", colour toggle: g_stHMI_EL4032EcSlaveStateBits.bPortA
    Rectangle (627,426 85x18), "Port B", colour toggle: g_stHMI_EL4032EcSlaveStateBits.bPortB
    Rectangle (627,446 85x18), "Port C", colour toggle: g_stHMI_EL4032EcSlaveStateBits.bPortC
    Rectangle (627,466 85x18), "Port D", colour toggle: g_stHMI_EL4032EcSlaveStateBits.bPortD
    Group (714,42 89x451)
        RoundedRectangle (0,2 89x449)
        Label (2,0 85x25), "EL7201 #1"
        Rectangle (2,19 85x22), "Sftw Rev: %s", text variable: g_iHMI_ProdCodeEL7201_1
        Rectangle (2,39 85x22), "Port A CRC: %s", text variable: g_stHMI_EL7201_1CrcErrorEx.portA
        Rectangle (2,59 85x22), "Port B CRC: %s", text variable: g_stHMI_EL7201_1CrcErrorEx.portB
        Rectangle (2,79 85x22), "Port C CRC: %s", text variable: g_stHMI_EL7201_1CrcErrorEx.portC
        Rectangle (2,99 85x22), "Port D CRC: %s", text variable: g_stHMI_EL7201_1CrcErrorEx.portD
        Rectangle (2,124 85x18), "BootStrap", colour toggle: g_stHMI_EL7201_1EcSlaveStateBits.bBootStrap
        Rectangle (2,144 85x18), "Init", colour toggle: g_stHMI_EL7201_1EcSlaveStateBits.bInit
        Rectangle (2,164 85x18), "PreOP", colour toggle: g_stHMI_EL7201_1EcSlaveStateBits.bPreop
        Rectangle (2,184 85x18), "SafeOP", colour toggle: g_stHMI_EL7201_1EcSlaveStateBits.bSafeOp
        Rectangle (2,204 85x18), "OP", colour toggle: g_stHMI_EL7201_1EcSlaveStateBits.bOp
        Rectangle (2,224 85x18), "Error", colour toggle: g_stHMI_EL7201_1EcSlaveStateBits.bError
        Rectangle (2,244 85x18), "InvVPRS", colour toggle: g_stHMI_EL7201_1EcSlaveStateBits.bInvVPRS
        Rectangle (2,264 85x18), "InitCmdError", colour toggle: g_stHMI_EL7201_1EcSlaveStateBits.bInitCmdError
        Rectangle (2,284 85x18), "LinkNotPresent", colour toggle: g_stHMI_EL7201_1EcSlaveStateBits.bLinkNotPresent
        Rectangle (2,304 85x18), "Link_w/o_Com", colour toggle: g_stHMI_EL7201_1EcSlaveStateBits.bLinkWithoutComm
        Rectangle (2,324 85x18), "LinkMissing", colour toggle: g_stHMI_EL7201_1EcSlaveStateBits.bLinkMissing
        Rectangle (2,344 85x18), "AdditionalLink", colour toggle: g_stHMI_EL7201_1EcSlaveStateBits.bAdditionalLink
        Rectangle (2,364 85x18), "Port A", colour toggle: g_stHMI_EL7201_1EcSlaveStateBits.bPortA
        Rectangle (2,384 85x18), "Port B", colour toggle: g_stHMI_EL7201_1EcSlaveStateBits.bPortB
        Rectangle (2,404 85x18), "Port C", colour toggle: g_stHMI_EL7201_1EcSlaveStateBits.bPortC
        Rectangle (2,424 85x18), "Port D", colour toggle: g_stHMI_EL7201_1EcSlaveStateBits.bPortD
    Group (803,42 89x451)
        RoundedRectangle (0,2 89x449)
        Label (2,0 85x25), "EL7201 #2"
        Rectangle (2,19 85x22), "Sftw Rev: %s", text variable: g_iHMI_ProdCodeEL7201_2
        Rectangle (2,39 85x22), "Port A CRC: %s", text variable: g_stHMI_EL7201_2CrcErrorEx.portA
        Rectangle (2,59 85x22), "Port B CRC: %s", text variable: g_stHMI_EL7201_2CrcErrorEx.portB
        Rectangle (2,79 85x22), "Port C CRC: %s", text variable: g_stHMI_EL7201_2CrcErrorEx.portC
        Rectangle (2,99 85x22), "Port D CRC: %s", text variable: g_stHMI_EL7201_2CrcErrorEx.portD
        Rectangle (2,124 85x18), "BootStrap", colour toggle: g_stHMI_EL7201_2EcSlaveStateBits.bBootStrap
        Rectangle (2,144 85x18), "Init", colour toggle: g_stHMI_EL7201_2EcSlaveStateBits.bInit
        Rectangle (2,164 85x18), "PreOP", colour toggle: g_stHMI_EL7201_2EcSlaveStateBits.bPreop
        Rectangle (2,184 85x18), "SafeOP", colour toggle: g_stHMI_EL7201_2EcSlaveStateBits.bSafeOp
        Rectangle (2,204 85x18), "OP", colour toggle: g_stHMI_EL7201_2EcSlaveStateBits.bOp
        Rectangle (2,224 85x18), "Error", colour toggle: g_stHMI_EL7201_2EcSlaveStateBits.bError
        Rectangle (2,244 85x18), "InvVPRS", colour toggle: g_stHMI_EL7201_2EcSlaveStateBits.bInvVPRS
        Rectangle (2,264 85x18), "InitCmdError", colour toggle: g_stHMI_EL7201_2EcSlaveStateBits.bInitCmdError
        Rectangle (2,284 85x18), "LinkNotPresent", colour toggle: g_stHMI_EL7201_2EcSlaveStateBits.bLinkNotPresent
        Rectangle (2,304 85x18), "Link_w/o_Com", colour toggle: g_stHMI_EL7201_2EcSlaveStateBits.bLinkWithoutComm
        Rectangle (2,324 85x18), "LinkMissing", colour toggle: g_stHMI_EL7201_2EcSlaveStateBits.bLinkMissing
        Rectangle (2,344 85x18), "AdditionalLink", colour toggle: g_stHMI_EL7201_2EcSlaveStateBits.bAdditionalLink
        Rectangle (2,364 85x18), "Port A", colour toggle: g_stHMI_EL7201_2EcSlaveStateBits.bPortA
        Rectangle (2,384 85x18), "Port B", colour toggle: g_stHMI_EL7201_2EcSlaveStateBits.bPortB
        Rectangle (2,404 85x18), "Port C", colour toggle: g_stHMI_EL7201_2EcSlaveStateBits.bPortC
        Rectangle (2,424 85x18), "Port D", colour toggle: g_stHMI_EL7201_2EcSlaveStateBits.bPortD
    Group (892,42 89x451)
        RoundedRectangle (0,2 89x449)
        Label (2,0 85x25), "EK1122"
        Rectangle (2,19 85x22), "Sftw Rev: %s", text variable: g_iHMI_ProdCodeEK1122
        Rectangle (2,39 85x22), "Port A CRC: %s", text variable: g_stHMI_EK1122_CrcErrorEx.portA
        Rectangle (2,59 85x22), "Port B CRC: %s", text variable: g_stHMI_EK1122_CrcErrorEx.portB
        Rectangle (2,79 85x22), "Port C CRC: %s", text variable: g_stHMI_EK1122_CrcErrorEx.portC
        Rectangle (2,99 85x22), "Port D CRC: %s", text variable: g_stHMI_EK1122_CrcErrorEx.portD
        Rectangle (2,124 85x18), "BootStrap", colour toggle: g_stHMI_EK1122_EcSlaveStateBits.bBootStrap
        Rectangle (2,144 85x18), "Init", colour toggle: g_stHMI_EK1122_EcSlaveStateBits.bInit
        Rectangle (2,164 85x18), "PreOP", colour toggle: g_stHMI_EK1122_EcSlaveStateBits.bPreop
        Rectangle (2,184 85x18), "SafeOP", colour toggle: g_stHMI_EK1122_EcSlaveStateBits.bSafeOp
        Rectangle (2,204 85x18), "OP", colour toggle: g_stHMI_EK1122_EcSlaveStateBits.bOp
        Rectangle (2,224 85x18), "Error", colour toggle: g_stHMI_EK1122_EcSlaveStateBits.bError
        Rectangle (2,244 85x18), "InvVPRS", colour toggle: g_stHMI_EK1122_EcSlaveStateBits.bInvVPRS
        Rectangle (2,264 85x18), "InitCmdError", colour toggle: g_stHMI_EK1122_EcSlaveStateBits.bInitCmdError
        Rectangle (2,284 85x18), "LinkNotPresent", colour toggle: g_stHMI_EK1122_EcSlaveStateBits.bLinkNotPresent
        Rectangle (2,304 85x18), "Link_w/o_Com", colour toggle: g_stHMI_EK1122_EcSlaveStateBits.bLinkWithoutComm
        Rectangle (2,324 85x18), "LinkMissing", colour toggle: g_stHMI_EK1122_EcSlaveStateBits.bLinkMissing
        Rectangle (2,344 85x18), "AdditionalLink", colour toggle: g_stHMI_EK1122_EcSlaveStateBits.bAdditionalLink
        Rectangle (2,364 85x18), "Port A", colour toggle: g_stHMI_EK1122_EcSlaveStateBits.bPortA
        Rectangle (2,384 85x18), "Port B", colour toggle: g_stHMI_EK1122_EcSlaveStateBits.bPortB
        Rectangle (2,404 85x18), "Port C", colour toggle: g_stHMI_EK1122_EcSlaveStateBits.bPortC
        Rectangle (2,424 85x18), "Port D", colour toggle: g_stHMI_EK1122_EcSlaveStateBits.bPortD
END_VISUALIZATION

